// TwinCAT 3 PLC project CSVExample
// ProgramVersion: 3.1.0.8
// libraries:
//   Tc2_Math, * (Beckhoff Automation GmbH)
//   Tc2_Standard, * (Beckhoff Automation GmbH)
//   Tc2_System, * (Beckhoff Automation GmbH)
//   Tc2_Utilities, * (Beckhoff Automation GmbH)
//   Tc3_Module, * (Beckhoff Automation GmbH)
//   VisuDialogs, * (System)
//   Base Interfaces,newest,System
//   VisuSymbols,3.5.10.0,System
// project tree:
//   DUTs/ arr_rt.TcDUT (not stored), ENUM_BufferMgmt.TcDUT, ENUM_SeqSM.TcDUT, ST_CSV_Record.TcDUT (not stored)
//   DUTs/typ_FB_Debounce/ typFBDInOut.TcDUT (not stored), typFBDInput.TcDUT, typFBDOutput.TcDUT (not stored), typ_FBInt_Debounce.TcDUT
//   DUTs/typ_FB_DMX/ ENUM_IQ_OpMode.TcDUT (not stored), ENUM_I_ValRange.TcDUT (not stored), ENUM_I_Waveform.TcDUT, typDMXInOut.TcDUT (not stored), typDMXInput.TcDUT, typDMXOutput.TcDUT, typ_FBInt_DMX.TcDUT
//   / GlobalTextList.TcGTLO, PlcTask.TcTTO, Visualization Manager.TcVMO (not stored)
//   GVLs/ gc.TcGVL, gFB.TcGVL, GVL.TcGVL, g_ast.TcGVL
//   POUs/CSV read_write in binary mode/ P_BinaryModeRead.TcPOU, P_BinaryModeWrite.TcPOU (not stored)
//   POUs/CSV read_write in text mode/ P_TextModeRead.TcPOU (not stored), P_TextModeWrite.TcPOU (not stored)
//   POUs/ DMXTest.TcPOU, MAIN.TcPOU, P_ArgToConvExample.TcPOU, P_StringToConvExample.TcPOU
//   POUs/FunctionBlocks/ FB_DMX.TcPOU, FB_InputDebounce.TcPOU (not stored)
//   POUs/FunctionBlocks/HelperPRG/ InterfaceLink.TcPOU, IOParams.TcPOU
//   POUs/Functions/ f_to_Period.TcPOU, Map.TcPOU, MapClamp.TcPOU, SclByteDMX.TcPOU (not stored), SclBytePNP.TcPOU
//   VISUs/ Visualization.TcVIS
// real-time tasks:
//   TASK PlcTask: cycle T#10ms, priority 20, ADS port 350
// I/O:
//   DEVICE Device 1 (EtherCAT) (disabled), AmsNetId 192.168.1.208.2.1
//     Term 1 (EK1100) [EK1100 EtherCAT Coupler (2A E-Bus)]
//       Term 2 (EL6851) [EL6851 DMX Master]
//       Term 3 (EL1008) [EL1008 8Ch. Dig. Input 24V, 3ms]
//       Term 4 (EL1008) [EL1008 8Ch. Dig. Input 24V, 3ms]
//       Term 5 (EL1008) [EL1008 8Ch. Dig. Input 24V, 3ms]
//       Term 29 (EL1008) [EL1008 8Ch. Dig. Input 24V, 3ms]
//       Term 30 (EL1008) [EL1008 8Ch. Dig. Input 24V, 3ms]
//       Term 31 (EL1008) [EL1008 8Ch. Dig. Input 24V, 3ms]
//       Term 32 (EL1008) [EL1008 8Ch. Dig. Input 24V, 3ms]
//       Term 33 (EL1008) [EL1008 8Ch. Dig. Input 24V, 3ms]
//       Term 34 (EL1008) [EL1008 8Ch. Dig. Input 24V, 3ms]
//       Term 35 (EL1008) [EL1008 8Ch. Dig. Input 24V, 3ms]
//       Term 36 (EL1088) [EL1088 8Ch. Dig. Input 24V, 3ms, negative]
//       Term 37 (EL1088) [EL1088 8Ch. Dig. Input 24V, 3ms, negative]
//       Term 38 (EL1088) [EL1088 8Ch. Dig. Input 24V, 3ms, negative]
//       Term 39 (EL1088) [EL1088 8Ch. Dig. Input 24V, 3ms, negative]
//       Term 40 (EL1088) [EL1088 8Ch. Dig. Input 24V, 3ms, negative]
//       Term 41 (EL9410) [EL9410 E-Bus Power Supplier  (Diagnostics)]
//       Term 42 (EL1088) [EL1088 8Ch. Dig. Input 24V, 3ms, negative]
//       Term 43 (EL1088) [EL1088 8Ch. Dig. Input 24V, 3ms, negative]
//       Term 44 (EL1088) [EL1088 8Ch. Dig. Input 24V, 3ms, negative]
//       Term 45 (EL1088) [EL1088 8Ch. Dig. Input 24V, 3ms, negative]
//       Term 46 (EL1088) [EL1088 8Ch. Dig. Input 24V, 3ms, negative]
//       Term 47 (EL9011) [EL9011 End Terminal]
// variable links:
//   CSVExample/CSVExample Instance <-> Device 1 (EtherCAT)/Term 1 (EK1100)/Term 2 (EL6851)
//     PlcTask Outputs/g_ast.DMXHWOut[0] <-> DMX Channel 1-64/Channel 1
//     PlcTask Outputs/g_ast.DMXHWOut[100] <-> DMX Channel 65-128/Channel 101
//     PlcTask Outputs/g_ast.DMXHWOut[101] <-> DMX Channel 65-128/Channel 102
//     PlcTask Outputs/g_ast.DMXHWOut[102] <-> DMX Channel 65-128/Channel 103
//     PlcTask Outputs/g_ast.DMXHWOut[103] <-> DMX Channel 65-128/Channel 104
//     PlcTask Outputs/g_ast.DMXHWOut[104] <-> DMX Channel 65-128/Channel 105
//     PlcTask Outputs/g_ast.DMXHWOut[105] <-> DMX Channel 65-128/Channel 106
//     PlcTask Outputs/g_ast.DMXHWOut[106] <-> DMX Channel 65-128/Channel 107
//     PlcTask Outputs/g_ast.DMXHWOut[107] <-> DMX Channel 65-128/Channel 108
//     PlcTask Outputs/g_ast.DMXHWOut[108] <-> DMX Channel 65-128/Channel 109
//     PlcTask Outputs/g_ast.DMXHWOut[109] <-> DMX Channel 65-128/Channel 110
//     PlcTask Outputs/g_ast.DMXHWOut[10] <-> DMX Channel 1-64/Channel 11
//     PlcTask Outputs/g_ast.DMXHWOut[110] <-> DMX Channel 65-128/Channel 111
//     PlcTask Outputs/g_ast.DMXHWOut[111] <-> DMX Channel 65-128/Channel 112
//     PlcTask Outputs/g_ast.DMXHWOut[112] <-> DMX Channel 65-128/Channel 113
//     PlcTask Outputs/g_ast.DMXHWOut[113] <-> DMX Channel 65-128/Channel 114
//     PlcTask Outputs/g_ast.DMXHWOut[114] <-> DMX Channel 65-128/Channel 115
//     PlcTask Outputs/g_ast.DMXHWOut[115] <-> DMX Channel 65-128/Channel 116
//     PlcTask Outputs/g_ast.DMXHWOut[116] <-> DMX Channel 65-128/Channel 117
//     PlcTask Outputs/g_ast.DMXHWOut[117] <-> DMX Channel 65-128/Channel 118
//     PlcTask Outputs/g_ast.DMXHWOut[118] <-> DMX Channel 65-128/Channel 119
//     PlcTask Outputs/g_ast.DMXHWOut[119] <-> DMX Channel 65-128/Channel 120
//     PlcTask Outputs/g_ast.DMXHWOut[11] <-> DMX Channel 1-64/Channel 12
//     PlcTask Outputs/g_ast.DMXHWOut[120] <-> DMX Channel 65-128/Channel 121
//     PlcTask Outputs/g_ast.DMXHWOut[121] <-> DMX Channel 65-128/Channel 122
//     PlcTask Outputs/g_ast.DMXHWOut[122] <-> DMX Channel 65-128/Channel 123
//     PlcTask Outputs/g_ast.DMXHWOut[123] <-> DMX Channel 65-128/Channel 124
//     PlcTask Outputs/g_ast.DMXHWOut[124] <-> DMX Channel 65-128/Channel 125
//     PlcTask Outputs/g_ast.DMXHWOut[125] <-> DMX Channel 65-128/Channel 126
//     PlcTask Outputs/g_ast.DMXHWOut[126] <-> DMX Channel 65-128/Channel 127
//     PlcTask Outputs/g_ast.DMXHWOut[127] <-> DMX Channel 65-128/Channel 128
//     PlcTask Outputs/g_ast.DMXHWOut[128] <-> DMX Channel 129-192/Channel 129
//     PlcTask Outputs/g_ast.DMXHWOut[129] <-> DMX Channel 129-192/Channel 130
//     PlcTask Outputs/g_ast.DMXHWOut[12] <-> DMX Channel 1-64/Channel 13
//     PlcTask Outputs/g_ast.DMXHWOut[130] <-> DMX Channel 129-192/Channel 131
//     PlcTask Outputs/g_ast.DMXHWOut[131] <-> DMX Channel 129-192/Channel 132
//     PlcTask Outputs/g_ast.DMXHWOut[132] <-> DMX Channel 129-192/Channel 133
//     PlcTask Outputs/g_ast.DMXHWOut[133] <-> DMX Channel 129-192/Channel 134
//     PlcTask Outputs/g_ast.DMXHWOut[134] <-> DMX Channel 129-192/Channel 135
//     PlcTask Outputs/g_ast.DMXHWOut[135] <-> DMX Channel 129-192/Channel 136
//     PlcTask Outputs/g_ast.DMXHWOut[136] <-> DMX Channel 129-192/Channel 137
//     PlcTask Outputs/g_ast.DMXHWOut[137] <-> DMX Channel 129-192/Channel 138
//     PlcTask Outputs/g_ast.DMXHWOut[138] <-> DMX Channel 129-192/Channel 139
//     PlcTask Outputs/g_ast.DMXHWOut[139] <-> DMX Channel 129-192/Channel 140
//     PlcTask Outputs/g_ast.DMXHWOut[13] <-> DMX Channel 1-64/Channel 14
//     PlcTask Outputs/g_ast.DMXHWOut[140] <-> DMX Channel 129-192/Channel 141
//     PlcTask Outputs/g_ast.DMXHWOut[141] <-> DMX Channel 129-192/Channel 142
//     PlcTask Outputs/g_ast.DMXHWOut[142] <-> DMX Channel 129-192/Channel 143
//     PlcTask Outputs/g_ast.DMXHWOut[143] <-> DMX Channel 129-192/Channel 144
//     PlcTask Outputs/g_ast.DMXHWOut[144] <-> DMX Channel 129-192/Channel 145
//     PlcTask Outputs/g_ast.DMXHWOut[145] <-> DMX Channel 129-192/Channel 146
//     PlcTask Outputs/g_ast.DMXHWOut[146] <-> DMX Channel 129-192/Channel 147
//     PlcTask Outputs/g_ast.DMXHWOut[147] <-> DMX Channel 129-192/Channel 148
//     PlcTask Outputs/g_ast.DMXHWOut[148] <-> DMX Channel 129-192/Channel 149
//     PlcTask Outputs/g_ast.DMXHWOut[149] <-> DMX Channel 129-192/Channel 150
//     PlcTask Outputs/g_ast.DMXHWOut[14] <-> DMX Channel 1-64/Channel 15
//     PlcTask Outputs/g_ast.DMXHWOut[150] <-> DMX Channel 129-192/Channel 151
//     PlcTask Outputs/g_ast.DMXHWOut[151] <-> DMX Channel 129-192/Channel 152
//     PlcTask Outputs/g_ast.DMXHWOut[152] <-> DMX Channel 129-192/Channel 153
//     PlcTask Outputs/g_ast.DMXHWOut[153] <-> DMX Channel 129-192/Channel 154
//     PlcTask Outputs/g_ast.DMXHWOut[154] <-> DMX Channel 129-192/Channel 155
//     PlcTask Outputs/g_ast.DMXHWOut[155] <-> DMX Channel 129-192/Channel 156
//     PlcTask Outputs/g_ast.DMXHWOut[156] <-> DMX Channel 129-192/Channel 157
//     PlcTask Outputs/g_ast.DMXHWOut[157] <-> DMX Channel 129-192/Channel 158
//     PlcTask Outputs/g_ast.DMXHWOut[158] <-> DMX Channel 129-192/Channel 159
//     PlcTask Outputs/g_ast.DMXHWOut[159] <-> DMX Channel 129-192/Channel 160
//     PlcTask Outputs/g_ast.DMXHWOut[15] <-> DMX Channel 1-64/Channel 16
//     PlcTask Outputs/g_ast.DMXHWOut[160] <-> DMX Channel 129-192/Channel 161
//     PlcTask Outputs/g_ast.DMXHWOut[161] <-> DMX Channel 129-192/Channel 162
//     PlcTask Outputs/g_ast.DMXHWOut[162] <-> DMX Channel 129-192/Channel 163
//     PlcTask Outputs/g_ast.DMXHWOut[163] <-> DMX Channel 129-192/Channel 164
//     PlcTask Outputs/g_ast.DMXHWOut[164] <-> DMX Channel 129-192/Channel 165
//     PlcTask Outputs/g_ast.DMXHWOut[165] <-> DMX Channel 129-192/Channel 166
//     PlcTask Outputs/g_ast.DMXHWOut[166] <-> DMX Channel 129-192/Channel 167
//     PlcTask Outputs/g_ast.DMXHWOut[167] <-> DMX Channel 129-192/Channel 168
//     PlcTask Outputs/g_ast.DMXHWOut[168] <-> DMX Channel 129-192/Channel 169
//     PlcTask Outputs/g_ast.DMXHWOut[169] <-> DMX Channel 129-192/Channel 170
//     PlcTask Outputs/g_ast.DMXHWOut[16] <-> DMX Channel 1-64/Channel 17
//     PlcTask Outputs/g_ast.DMXHWOut[170] <-> DMX Channel 129-192/Channel 171
//     PlcTask Outputs/g_ast.DMXHWOut[171] <-> DMX Channel 129-192/Channel 172
//     PlcTask Outputs/g_ast.DMXHWOut[172] <-> DMX Channel 129-192/Channel 173
//     PlcTask Outputs/g_ast.DMXHWOut[173] <-> DMX Channel 129-192/Channel 174
//     PlcTask Outputs/g_ast.DMXHWOut[174] <-> DMX Channel 129-192/Channel 175
//     PlcTask Outputs/g_ast.DMXHWOut[175] <-> DMX Channel 129-192/Channel 176
//     PlcTask Outputs/g_ast.DMXHWOut[176] <-> DMX Channel 129-192/Channel 177
//     PlcTask Outputs/g_ast.DMXHWOut[177] <-> DMX Channel 129-192/Channel 178
//     PlcTask Outputs/g_ast.DMXHWOut[178] <-> DMX Channel 129-192/Channel 179
//     PlcTask Outputs/g_ast.DMXHWOut[179] <-> DMX Channel 129-192/Channel 180
//     PlcTask Outputs/g_ast.DMXHWOut[17] <-> DMX Channel 1-64/Channel 18
//     PlcTask Outputs/g_ast.DMXHWOut[180] <-> DMX Channel 129-192/Channel 181
//     PlcTask Outputs/g_ast.DMXHWOut[181] <-> DMX Channel 129-192/Channel 182
//     PlcTask Outputs/g_ast.DMXHWOut[182] <-> DMX Channel 129-192/Channel 183
//     PlcTask Outputs/g_ast.DMXHWOut[183] <-> DMX Channel 129-192/Channel 184
//     PlcTask Outputs/g_ast.DMXHWOut[184] <-> DMX Channel 129-192/Channel 185
//     PlcTask Outputs/g_ast.DMXHWOut[185] <-> DMX Channel 129-192/Channel 186
//     PlcTask Outputs/g_ast.DMXHWOut[186] <-> DMX Channel 129-192/Channel 187
//     PlcTask Outputs/g_ast.DMXHWOut[187] <-> DMX Channel 129-192/Channel 188
//     PlcTask Outputs/g_ast.DMXHWOut[188] <-> DMX Channel 129-192/Channel 189
//     PlcTask Outputs/g_ast.DMXHWOut[189] <-> DMX Channel 129-192/Channel 190
//     PlcTask Outputs/g_ast.DMXHWOut[18] <-> DMX Channel 1-64/Channel 19
//     PlcTask Outputs/g_ast.DMXHWOut[190] <-> DMX Channel 129-192/Channel 191
//     PlcTask Outputs/g_ast.DMXHWOut[191] <-> DMX Channel 129-192/Channel 192
//     PlcTask Outputs/g_ast.DMXHWOut[192] <-> DMX Channel 193-256/Channel 193
//     PlcTask Outputs/g_ast.DMXHWOut[193] <-> DMX Channel 193-256/Channel 194
//     PlcTask Outputs/g_ast.DMXHWOut[194] <-> DMX Channel 193-256/Channel 195
//     PlcTask Outputs/g_ast.DMXHWOut[195] <-> DMX Channel 193-256/Channel 196
//     PlcTask Outputs/g_ast.DMXHWOut[196] <-> DMX Channel 193-256/Channel 197
//     PlcTask Outputs/g_ast.DMXHWOut[197] <-> DMX Channel 193-256/Channel 198
//     PlcTask Outputs/g_ast.DMXHWOut[198] <-> DMX Channel 193-256/Channel 199
//     PlcTask Outputs/g_ast.DMXHWOut[199] <-> DMX Channel 193-256/Channel 200
//     PlcTask Outputs/g_ast.DMXHWOut[19] <-> DMX Channel 1-64/Channel 20
//     PlcTask Outputs/g_ast.DMXHWOut[1] <-> DMX Channel 1-64/Channel 2
//     PlcTask Outputs/g_ast.DMXHWOut[200] <-> DMX Channel 193-256/Channel 201
//     PlcTask Outputs/g_ast.DMXHWOut[201] <-> DMX Channel 193-256/Channel 202
//     PlcTask Outputs/g_ast.DMXHWOut[202] <-> DMX Channel 193-256/Channel 203
//     PlcTask Outputs/g_ast.DMXHWOut[203] <-> DMX Channel 193-256/Channel 204
//     PlcTask Outputs/g_ast.DMXHWOut[204] <-> DMX Channel 193-256/Channel 205
//     PlcTask Outputs/g_ast.DMXHWOut[205] <-> DMX Channel 193-256/Channel 206
//     PlcTask Outputs/g_ast.DMXHWOut[206] <-> DMX Channel 193-256/Channel 207
//     PlcTask Outputs/g_ast.DMXHWOut[207] <-> DMX Channel 193-256/Channel 208
//     PlcTask Outputs/g_ast.DMXHWOut[208] <-> DMX Channel 193-256/Channel 209
//     PlcTask Outputs/g_ast.DMXHWOut[209] <-> DMX Channel 193-256/Channel 210
//     PlcTask Outputs/g_ast.DMXHWOut[20] <-> DMX Channel 1-64/Channel 21
//     PlcTask Outputs/g_ast.DMXHWOut[210] <-> DMX Channel 193-256/Channel 211
//     PlcTask Outputs/g_ast.DMXHWOut[211] <-> DMX Channel 193-256/Channel 212
//     PlcTask Outputs/g_ast.DMXHWOut[212] <-> DMX Channel 193-256/Channel 213
//     PlcTask Outputs/g_ast.DMXHWOut[213] <-> DMX Channel 193-256/Channel 214
//     PlcTask Outputs/g_ast.DMXHWOut[214] <-> DMX Channel 193-256/Channel 215
//     PlcTask Outputs/g_ast.DMXHWOut[215] <-> DMX Channel 193-256/Channel 216
//     PlcTask Outputs/g_ast.DMXHWOut[216] <-> DMX Channel 193-256/Channel 217
//     PlcTask Outputs/g_ast.DMXHWOut[217] <-> DMX Channel 193-256/Channel 218
//     PlcTask Outputs/g_ast.DMXHWOut[218] <-> DMX Channel 193-256/Channel 219
//     PlcTask Outputs/g_ast.DMXHWOut[219] <-> DMX Channel 193-256/Channel 220
//     PlcTask Outputs/g_ast.DMXHWOut[21] <-> DMX Channel 1-64/Channel 22
//     PlcTask Outputs/g_ast.DMXHWOut[220] <-> DMX Channel 193-256/Channel 221
//     PlcTask Outputs/g_ast.DMXHWOut[221] <-> DMX Channel 193-256/Channel 222
//     PlcTask Outputs/g_ast.DMXHWOut[222] <-> DMX Channel 193-256/Channel 223
//     PlcTask Outputs/g_ast.DMXHWOut[223] <-> DMX Channel 193-256/Channel 224
//     PlcTask Outputs/g_ast.DMXHWOut[224] <-> DMX Channel 193-256/Channel 225
//     PlcTask Outputs/g_ast.DMXHWOut[225] <-> DMX Channel 193-256/Channel 226
//     PlcTask Outputs/g_ast.DMXHWOut[226] <-> DMX Channel 193-256/Channel 227
//     PlcTask Outputs/g_ast.DMXHWOut[227] <-> DMX Channel 193-256/Channel 228
//     PlcTask Outputs/g_ast.DMXHWOut[228] <-> DMX Channel 193-256/Channel 229
//     PlcTask Outputs/g_ast.DMXHWOut[229] <-> DMX Channel 193-256/Channel 230
//     PlcTask Outputs/g_ast.DMXHWOut[22] <-> DMX Channel 1-64/Channel 23
//     PlcTask Outputs/g_ast.DMXHWOut[230] <-> DMX Channel 193-256/Channel 231
//     PlcTask Outputs/g_ast.DMXHWOut[231] <-> DMX Channel 193-256/Channel 232
//     PlcTask Outputs/g_ast.DMXHWOut[232] <-> DMX Channel 193-256/Channel 233
//     PlcTask Outputs/g_ast.DMXHWOut[233] <-> DMX Channel 193-256/Channel 234
//     PlcTask Outputs/g_ast.DMXHWOut[234] <-> DMX Channel 193-256/Channel 235
//     PlcTask Outputs/g_ast.DMXHWOut[235] <-> DMX Channel 193-256/Channel 236
//     PlcTask Outputs/g_ast.DMXHWOut[236] <-> DMX Channel 193-256/Channel 237
//     PlcTask Outputs/g_ast.DMXHWOut[237] <-> DMX Channel 193-256/Channel 238
//     PlcTask Outputs/g_ast.DMXHWOut[238] <-> DMX Channel 193-256/Channel 239
//     PlcTask Outputs/g_ast.DMXHWOut[239] <-> DMX Channel 193-256/Channel 240
//     PlcTask Outputs/g_ast.DMXHWOut[23] <-> DMX Channel 1-64/Channel 24
//     PlcTask Outputs/g_ast.DMXHWOut[240] <-> DMX Channel 193-256/Channel 241
//     PlcTask Outputs/g_ast.DMXHWOut[241] <-> DMX Channel 193-256/Channel 242
//     PlcTask Outputs/g_ast.DMXHWOut[242] <-> DMX Channel 193-256/Channel 243
//     PlcTask Outputs/g_ast.DMXHWOut[243] <-> DMX Channel 193-256/Channel 244
//     PlcTask Outputs/g_ast.DMXHWOut[244] <-> DMX Channel 193-256/Channel 245
//     PlcTask Outputs/g_ast.DMXHWOut[245] <-> DMX Channel 193-256/Channel 246
//     PlcTask Outputs/g_ast.DMXHWOut[246] <-> DMX Channel 193-256/Channel 247
//     PlcTask Outputs/g_ast.DMXHWOut[247] <-> DMX Channel 193-256/Channel 248
//     PlcTask Outputs/g_ast.DMXHWOut[248] <-> DMX Channel 193-256/Channel 249
//     PlcTask Outputs/g_ast.DMXHWOut[249] <-> DMX Channel 193-256/Channel 250
//     PlcTask Outputs/g_ast.DMXHWOut[24] <-> DMX Channel 1-64/Channel 25
//     PlcTask Outputs/g_ast.DMXHWOut[250] <-> DMX Channel 193-256/Channel 251
//     PlcTask Outputs/g_ast.DMXHWOut[251] <-> DMX Channel 193-256/Channel 252
//     PlcTask Outputs/g_ast.DMXHWOut[252] <-> DMX Channel 193-256/Channel 253
//     PlcTask Outputs/g_ast.DMXHWOut[253] <-> DMX Channel 193-256/Channel 254
//     PlcTask Outputs/g_ast.DMXHWOut[254] <-> DMX Channel 193-256/Channel 255
//     PlcTask Outputs/g_ast.DMXHWOut[255] <-> DMX Channel 193-256/Channel 256
//     PlcTask Outputs/g_ast.DMXHWOut[256] <-> DMX Channel 257-320/Channel 257
//     PlcTask Outputs/g_ast.DMXHWOut[257] <-> DMX Channel 257-320/Channel 258
//     PlcTask Outputs/g_ast.DMXHWOut[258] <-> DMX Channel 257-320/Channel 259
//     PlcTask Outputs/g_ast.DMXHWOut[259] <-> DMX Channel 257-320/Channel 260
//     PlcTask Outputs/g_ast.DMXHWOut[25] <-> DMX Channel 1-64/Channel 26
//     PlcTask Outputs/g_ast.DMXHWOut[260] <-> DMX Channel 257-320/Channel 261
//     PlcTask Outputs/g_ast.DMXHWOut[261] <-> DMX Channel 257-320/Channel 262
//     PlcTask Outputs/g_ast.DMXHWOut[262] <-> DMX Channel 257-320/Channel 263
//     PlcTask Outputs/g_ast.DMXHWOut[263] <-> DMX Channel 257-320/Channel 264
//     PlcTask Outputs/g_ast.DMXHWOut[264] <-> DMX Channel 257-320/Channel 265
//     PlcTask Outputs/g_ast.DMXHWOut[265] <-> DMX Channel 257-320/Channel 266
//     PlcTask Outputs/g_ast.DMXHWOut[266] <-> DMX Channel 257-320/Channel 267
//     PlcTask Outputs/g_ast.DMXHWOut[267] <-> DMX Channel 257-320/Channel 268
//     PlcTask Outputs/g_ast.DMXHWOut[268] <-> DMX Channel 257-320/Channel 269
//     PlcTask Outputs/g_ast.DMXHWOut[269] <-> DMX Channel 257-320/Channel 270
//     PlcTask Outputs/g_ast.DMXHWOut[26] <-> DMX Channel 1-64/Channel 27
//     PlcTask Outputs/g_ast.DMXHWOut[270] <-> DMX Channel 257-320/Channel 271
//     PlcTask Outputs/g_ast.DMXHWOut[271] <-> DMX Channel 257-320/Channel 272
//     PlcTask Outputs/g_ast.DMXHWOut[272] <-> DMX Channel 257-320/Channel 273
//     PlcTask Outputs/g_ast.DMXHWOut[273] <-> DMX Channel 257-320/Channel 274
//     PlcTask Outputs/g_ast.DMXHWOut[274] <-> DMX Channel 257-320/Channel 275
//     PlcTask Outputs/g_ast.DMXHWOut[275] <-> DMX Channel 257-320/Channel 276
//     PlcTask Outputs/g_ast.DMXHWOut[276] <-> DMX Channel 257-320/Channel 277
//     PlcTask Outputs/g_ast.DMXHWOut[277] <-> DMX Channel 257-320/Channel 278
//     PlcTask Outputs/g_ast.DMXHWOut[278] <-> DMX Channel 257-320/Channel 279
//     PlcTask Outputs/g_ast.DMXHWOut[279] <-> DMX Channel 257-320/Channel 280
//     PlcTask Outputs/g_ast.DMXHWOut[27] <-> DMX Channel 1-64/Channel 28
//     PlcTask Outputs/g_ast.DMXHWOut[280] <-> DMX Channel 257-320/Channel 281
//     PlcTask Outputs/g_ast.DMXHWOut[281] <-> DMX Channel 257-320/Channel 282
//     PlcTask Outputs/g_ast.DMXHWOut[282] <-> DMX Channel 257-320/Channel 283
//     PlcTask Outputs/g_ast.DMXHWOut[283] <-> DMX Channel 257-320/Channel 284
//     PlcTask Outputs/g_ast.DMXHWOut[284] <-> DMX Channel 257-320/Channel 285
//     PlcTask Outputs/g_ast.DMXHWOut[285] <-> DMX Channel 257-320/Channel 286
//     PlcTask Outputs/g_ast.DMXHWOut[286] <-> DMX Channel 257-320/Channel 287
//     PlcTask Outputs/g_ast.DMXHWOut[287] <-> DMX Channel 257-320/Channel 288
//     PlcTask Outputs/g_ast.DMXHWOut[288] <-> DMX Channel 257-320/Channel 289
//     PlcTask Outputs/g_ast.DMXHWOut[289] <-> DMX Channel 257-320/Channel 290
//     PlcTask Outputs/g_ast.DMXHWOut[28] <-> DMX Channel 1-64/Channel 29
//     PlcTask Outputs/g_ast.DMXHWOut[290] <-> DMX Channel 257-320/Channel 291
//     PlcTask Outputs/g_ast.DMXHWOut[291] <-> DMX Channel 257-320/Channel 292
//     PlcTask Outputs/g_ast.DMXHWOut[292] <-> DMX Channel 257-320/Channel 293
//     PlcTask Outputs/g_ast.DMXHWOut[293] <-> DMX Channel 257-320/Channel 294
//     PlcTask Outputs/g_ast.DMXHWOut[294] <-> DMX Channel 257-320/Channel 295
//     PlcTask Outputs/g_ast.DMXHWOut[295] <-> DMX Channel 257-320/Channel 296
//     PlcTask Outputs/g_ast.DMXHWOut[296] <-> DMX Channel 257-320/Channel 297
//     PlcTask Outputs/g_ast.DMXHWOut[297] <-> DMX Channel 257-320/Channel 298
//     PlcTask Outputs/g_ast.DMXHWOut[298] <-> DMX Channel 257-320/Channel 299
//     PlcTask Outputs/g_ast.DMXHWOut[299] <-> DMX Channel 257-320/Channel 300
//     PlcTask Outputs/g_ast.DMXHWOut[29] <-> DMX Channel 1-64/Channel 30
//     PlcTask Outputs/g_ast.DMXHWOut[2] <-> DMX Channel 1-64/Channel 3
//     PlcTask Outputs/g_ast.DMXHWOut[300] <-> DMX Channel 257-320/Channel 301
//     PlcTask Outputs/g_ast.DMXHWOut[301] <-> DMX Channel 257-320/Channel 302
//     PlcTask Outputs/g_ast.DMXHWOut[302] <-> DMX Channel 257-320/Channel 303
//     PlcTask Outputs/g_ast.DMXHWOut[303] <-> DMX Channel 257-320/Channel 304
//     PlcTask Outputs/g_ast.DMXHWOut[304] <-> DMX Channel 257-320/Channel 305
//     PlcTask Outputs/g_ast.DMXHWOut[305] <-> DMX Channel 257-320/Channel 306
//     PlcTask Outputs/g_ast.DMXHWOut[306] <-> DMX Channel 257-320/Channel 307
//     PlcTask Outputs/g_ast.DMXHWOut[307] <-> DMX Channel 257-320/Channel 308
//     PlcTask Outputs/g_ast.DMXHWOut[308] <-> DMX Channel 257-320/Channel 309
//     PlcTask Outputs/g_ast.DMXHWOut[309] <-> DMX Channel 257-320/Channel 310
//     PlcTask Outputs/g_ast.DMXHWOut[30] <-> DMX Channel 1-64/Channel 31
//     PlcTask Outputs/g_ast.DMXHWOut[310] <-> DMX Channel 257-320/Channel 311
//     PlcTask Outputs/g_ast.DMXHWOut[311] <-> DMX Channel 257-320/Channel 312
//     PlcTask Outputs/g_ast.DMXHWOut[312] <-> DMX Channel 257-320/Channel 313
//     PlcTask Outputs/g_ast.DMXHWOut[313] <-> DMX Channel 257-320/Channel 314
//     PlcTask Outputs/g_ast.DMXHWOut[314] <-> DMX Channel 257-320/Channel 315
//     PlcTask Outputs/g_ast.DMXHWOut[315] <-> DMX Channel 257-320/Channel 316
//     PlcTask Outputs/g_ast.DMXHWOut[316] <-> DMX Channel 257-320/Channel 317
//     PlcTask Outputs/g_ast.DMXHWOut[317] <-> DMX Channel 257-320/Channel 318
//     PlcTask Outputs/g_ast.DMXHWOut[318] <-> DMX Channel 257-320/Channel 319
//     PlcTask Outputs/g_ast.DMXHWOut[319] <-> DMX Channel 257-320/Channel 320
//     PlcTask Outputs/g_ast.DMXHWOut[31] <-> DMX Channel 1-64/Channel 32
//     PlcTask Outputs/g_ast.DMXHWOut[320] <-> DMX Channel 321-384/Channel 321
//     PlcTask Outputs/g_ast.DMXHWOut[321] <-> DMX Channel 321-384/Channel 322
//     PlcTask Outputs/g_ast.DMXHWOut[322] <-> DMX Channel 321-384/Channel 323
//     PlcTask Outputs/g_ast.DMXHWOut[323] <-> DMX Channel 321-384/Channel 324
//     PlcTask Outputs/g_ast.DMXHWOut[324] <-> DMX Channel 321-384/Channel 325
//     PlcTask Outputs/g_ast.DMXHWOut[325] <-> DMX Channel 321-384/Channel 326
//     PlcTask Outputs/g_ast.DMXHWOut[326] <-> DMX Channel 321-384/Channel 327
//     PlcTask Outputs/g_ast.DMXHWOut[327] <-> DMX Channel 321-384/Channel 328
//     PlcTask Outputs/g_ast.DMXHWOut[328] <-> DMX Channel 321-384/Channel 329
//     PlcTask Outputs/g_ast.DMXHWOut[329] <-> DMX Channel 321-384/Channel 330
//     PlcTask Outputs/g_ast.DMXHWOut[32] <-> DMX Channel 1-64/Channel 33
//     PlcTask Outputs/g_ast.DMXHWOut[330] <-> DMX Channel 321-384/Channel 331
//     PlcTask Outputs/g_ast.DMXHWOut[331] <-> DMX Channel 321-384/Channel 332
//     PlcTask Outputs/g_ast.DMXHWOut[332] <-> DMX Channel 321-384/Channel 333
//     PlcTask Outputs/g_ast.DMXHWOut[333] <-> DMX Channel 321-384/Channel 334
//     PlcTask Outputs/g_ast.DMXHWOut[334] <-> DMX Channel 321-384/Channel 335
//     PlcTask Outputs/g_ast.DMXHWOut[335] <-> DMX Channel 321-384/Channel 336
//     PlcTask Outputs/g_ast.DMXHWOut[336] <-> DMX Channel 321-384/Channel 337
//     PlcTask Outputs/g_ast.DMXHWOut[337] <-> DMX Channel 321-384/Channel 338
//     PlcTask Outputs/g_ast.DMXHWOut[338] <-> DMX Channel 321-384/Channel 339
//     PlcTask Outputs/g_ast.DMXHWOut[339] <-> DMX Channel 321-384/Channel 340
//     PlcTask Outputs/g_ast.DMXHWOut[33] <-> DMX Channel 1-64/Channel 34
//     PlcTask Outputs/g_ast.DMXHWOut[340] <-> DMX Channel 321-384/Channel 341
//     PlcTask Outputs/g_ast.DMXHWOut[341] <-> DMX Channel 321-384/Channel 342
//     PlcTask Outputs/g_ast.DMXHWOut[342] <-> DMX Channel 321-384/Channel 343
//     PlcTask Outputs/g_ast.DMXHWOut[343] <-> DMX Channel 321-384/Channel 344
//     PlcTask Outputs/g_ast.DMXHWOut[344] <-> DMX Channel 321-384/Channel 345
//     PlcTask Outputs/g_ast.DMXHWOut[345] <-> DMX Channel 321-384/Channel 346
//     PlcTask Outputs/g_ast.DMXHWOut[346] <-> DMX Channel 321-384/Channel 347
//     PlcTask Outputs/g_ast.DMXHWOut[347] <-> DMX Channel 321-384/Channel 348
//     PlcTask Outputs/g_ast.DMXHWOut[348] <-> DMX Channel 321-384/Channel 349
//     PlcTask Outputs/g_ast.DMXHWOut[349] <-> DMX Channel 321-384/Channel 350
//     PlcTask Outputs/g_ast.DMXHWOut[34] <-> DMX Channel 1-64/Channel 35
//     PlcTask Outputs/g_ast.DMXHWOut[350] <-> DMX Channel 321-384/Channel 351
//     PlcTask Outputs/g_ast.DMXHWOut[351] <-> DMX Channel 321-384/Channel 352
//     PlcTask Outputs/g_ast.DMXHWOut[352] <-> DMX Channel 321-384/Channel 353
//     PlcTask Outputs/g_ast.DMXHWOut[353] <-> DMX Channel 321-384/Channel 354
//     PlcTask Outputs/g_ast.DMXHWOut[354] <-> DMX Channel 321-384/Channel 355
//     PlcTask Outputs/g_ast.DMXHWOut[355] <-> DMX Channel 321-384/Channel 356
//     PlcTask Outputs/g_ast.DMXHWOut[356] <-> DMX Channel 321-384/Channel 357
//     PlcTask Outputs/g_ast.DMXHWOut[357] <-> DMX Channel 321-384/Channel 358
//     PlcTask Outputs/g_ast.DMXHWOut[358] <-> DMX Channel 321-384/Channel 359
//     PlcTask Outputs/g_ast.DMXHWOut[359] <-> DMX Channel 321-384/Channel 360
//     PlcTask Outputs/g_ast.DMXHWOut[35] <-> DMX Channel 1-64/Channel 36
//     PlcTask Outputs/g_ast.DMXHWOut[360] <-> DMX Channel 321-384/Channel 361
//     PlcTask Outputs/g_ast.DMXHWOut[361] <-> DMX Channel 321-384/Channel 362
//     PlcTask Outputs/g_ast.DMXHWOut[362] <-> DMX Channel 321-384/Channel 363
//     PlcTask Outputs/g_ast.DMXHWOut[363] <-> DMX Channel 321-384/Channel 364
//     PlcTask Outputs/g_ast.DMXHWOut[364] <-> DMX Channel 321-384/Channel 365
//     PlcTask Outputs/g_ast.DMXHWOut[365] <-> DMX Channel 321-384/Channel 366
//     PlcTask Outputs/g_ast.DMXHWOut[366] <-> DMX Channel 321-384/Channel 367
//     PlcTask Outputs/g_ast.DMXHWOut[367] <-> DMX Channel 321-384/Channel 368
//     PlcTask Outputs/g_ast.DMXHWOut[368] <-> DMX Channel 321-384/Channel 369
//     PlcTask Outputs/g_ast.DMXHWOut[369] <-> DMX Channel 321-384/Channel 370
//     PlcTask Outputs/g_ast.DMXHWOut[36] <-> DMX Channel 1-64/Channel 37
//     PlcTask Outputs/g_ast.DMXHWOut[370] <-> DMX Channel 321-384/Channel 371
//     PlcTask Outputs/g_ast.DMXHWOut[371] <-> DMX Channel 321-384/Channel 372
//     PlcTask Outputs/g_ast.DMXHWOut[372] <-> DMX Channel 321-384/Channel 373
//     PlcTask Outputs/g_ast.DMXHWOut[373] <-> DMX Channel 321-384/Channel 374
//     PlcTask Outputs/g_ast.DMXHWOut[374] <-> DMX Channel 321-384/Channel 375
//     PlcTask Outputs/g_ast.DMXHWOut[375] <-> DMX Channel 321-384/Channel 376
//     PlcTask Outputs/g_ast.DMXHWOut[376] <-> DMX Channel 321-384/Channel 377
//     PlcTask Outputs/g_ast.DMXHWOut[377] <-> DMX Channel 321-384/Channel 378
//     PlcTask Outputs/g_ast.DMXHWOut[378] <-> DMX Channel 321-384/Channel 379
//     PlcTask Outputs/g_ast.DMXHWOut[379] <-> DMX Channel 321-384/Channel 380
//     PlcTask Outputs/g_ast.DMXHWOut[37] <-> DMX Channel 1-64/Channel 38
//     PlcTask Outputs/g_ast.DMXHWOut[380] <-> DMX Channel 321-384/Channel 381
//     PlcTask Outputs/g_ast.DMXHWOut[381] <-> DMX Channel 321-384/Channel 382
//     PlcTask Outputs/g_ast.DMXHWOut[382] <-> DMX Channel 321-384/Channel 383
//     PlcTask Outputs/g_ast.DMXHWOut[383] <-> DMX Channel 321-384/Channel 384
//     PlcTask Outputs/g_ast.DMXHWOut[384] <-> DMX Channel 385-448/Channel 385
//     PlcTask Outputs/g_ast.DMXHWOut[385] <-> DMX Channel 385-448/Channel 386
//     PlcTask Outputs/g_ast.DMXHWOut[386] <-> DMX Channel 385-448/Channel 387
//     PlcTask Outputs/g_ast.DMXHWOut[387] <-> DMX Channel 385-448/Channel 388
//     PlcTask Outputs/g_ast.DMXHWOut[388] <-> DMX Channel 385-448/Channel 389
//     PlcTask Outputs/g_ast.DMXHWOut[389] <-> DMX Channel 385-448/Channel 390
//     PlcTask Outputs/g_ast.DMXHWOut[38] <-> DMX Channel 1-64/Channel 39
//     PlcTask Outputs/g_ast.DMXHWOut[390] <-> DMX Channel 385-448/Channel 391
//     PlcTask Outputs/g_ast.DMXHWOut[391] <-> DMX Channel 385-448/Channel 392
//     PlcTask Outputs/g_ast.DMXHWOut[392] <-> DMX Channel 385-448/Channel 393
//     PlcTask Outputs/g_ast.DMXHWOut[393] <-> DMX Channel 385-448/Channel 394
//     PlcTask Outputs/g_ast.DMXHWOut[394] <-> DMX Channel 385-448/Channel 395
//     PlcTask Outputs/g_ast.DMXHWOut[395] <-> DMX Channel 385-448/Channel 396
//     PlcTask Outputs/g_ast.DMXHWOut[396] <-> DMX Channel 385-448/Channel 397
//     PlcTask Outputs/g_ast.DMXHWOut[397] <-> DMX Channel 385-448/Channel 398
//     PlcTask Outputs/g_ast.DMXHWOut[398] <-> DMX Channel 385-448/Channel 399
//     PlcTask Outputs/g_ast.DMXHWOut[399] <-> DMX Channel 385-448/Channel 400
//     PlcTask Outputs/g_ast.DMXHWOut[39] <-> DMX Channel 1-64/Channel 40
//     PlcTask Outputs/g_ast.DMXHWOut[3] <-> DMX Channel 1-64/Channel 4
//     PlcTask Outputs/g_ast.DMXHWOut[400] <-> DMX Channel 385-448/Channel 401
//     PlcTask Outputs/g_ast.DMXHWOut[401] <-> DMX Channel 385-448/Channel 402
//     PlcTask Outputs/g_ast.DMXHWOut[402] <-> DMX Channel 385-448/Channel 403
//     PlcTask Outputs/g_ast.DMXHWOut[403] <-> DMX Channel 385-448/Channel 404
//     PlcTask Outputs/g_ast.DMXHWOut[404] <-> DMX Channel 385-448/Channel 405
//     PlcTask Outputs/g_ast.DMXHWOut[405] <-> DMX Channel 385-448/Channel 406
//     PlcTask Outputs/g_ast.DMXHWOut[406] <-> DMX Channel 385-448/Channel 407
//     PlcTask Outputs/g_ast.DMXHWOut[407] <-> DMX Channel 385-448/Channel 408
//     PlcTask Outputs/g_ast.DMXHWOut[408] <-> DMX Channel 385-448/Channel 409
//     PlcTask Outputs/g_ast.DMXHWOut[409] <-> DMX Channel 385-448/Channel 410
//     PlcTask Outputs/g_ast.DMXHWOut[40] <-> DMX Channel 1-64/Channel 41
//     PlcTask Outputs/g_ast.DMXHWOut[410] <-> DMX Channel 385-448/Channel 411
//     PlcTask Outputs/g_ast.DMXHWOut[411] <-> DMX Channel 385-448/Channel 412
//     PlcTask Outputs/g_ast.DMXHWOut[412] <-> DMX Channel 385-448/Channel 413
//     PlcTask Outputs/g_ast.DMXHWOut[413] <-> DMX Channel 385-448/Channel 414
//     PlcTask Outputs/g_ast.DMXHWOut[414] <-> DMX Channel 385-448/Channel 415
//     PlcTask Outputs/g_ast.DMXHWOut[415] <-> DMX Channel 385-448/Channel 416
//     PlcTask Outputs/g_ast.DMXHWOut[416] <-> DMX Channel 385-448/Channel 417
//     PlcTask Outputs/g_ast.DMXHWOut[417] <-> DMX Channel 385-448/Channel 418
//     PlcTask Outputs/g_ast.DMXHWOut[418] <-> DMX Channel 385-448/Channel 419
//     PlcTask Outputs/g_ast.DMXHWOut[419] <-> DMX Channel 385-448/Channel 420
//     PlcTask Outputs/g_ast.DMXHWOut[41] <-> DMX Channel 1-64/Channel 42
//     PlcTask Outputs/g_ast.DMXHWOut[420] <-> DMX Channel 385-448/Channel 421
//     PlcTask Outputs/g_ast.DMXHWOut[421] <-> DMX Channel 385-448/Channel 422
//     PlcTask Outputs/g_ast.DMXHWOut[422] <-> DMX Channel 385-448/Channel 423
//     PlcTask Outputs/g_ast.DMXHWOut[423] <-> DMX Channel 385-448/Channel 424
//     PlcTask Outputs/g_ast.DMXHWOut[424] <-> DMX Channel 385-448/Channel 425
//     PlcTask Outputs/g_ast.DMXHWOut[425] <-> DMX Channel 385-448/Channel 426
//     PlcTask Outputs/g_ast.DMXHWOut[426] <-> DMX Channel 385-448/Channel 427
//     PlcTask Outputs/g_ast.DMXHWOut[427] <-> DMX Channel 385-448/Channel 428
//     PlcTask Outputs/g_ast.DMXHWOut[428] <-> DMX Channel 385-448/Channel 429
//     PlcTask Outputs/g_ast.DMXHWOut[429] <-> DMX Channel 385-448/Channel 430
//     PlcTask Outputs/g_ast.DMXHWOut[42] <-> DMX Channel 1-64/Channel 43
//     PlcTask Outputs/g_ast.DMXHWOut[430] <-> DMX Channel 385-448/Channel 431
//     PlcTask Outputs/g_ast.DMXHWOut[431] <-> DMX Channel 385-448/Channel 432
//     PlcTask Outputs/g_ast.DMXHWOut[432] <-> DMX Channel 385-448/Channel 433
//     PlcTask Outputs/g_ast.DMXHWOut[433] <-> DMX Channel 385-448/Channel 434
//     PlcTask Outputs/g_ast.DMXHWOut[434] <-> DMX Channel 385-448/Channel 435
//     PlcTask Outputs/g_ast.DMXHWOut[435] <-> DMX Channel 385-448/Channel 436
//     PlcTask Outputs/g_ast.DMXHWOut[436] <-> DMX Channel 385-448/Channel 437
//     PlcTask Outputs/g_ast.DMXHWOut[437] <-> DMX Channel 385-448/Channel 438
//     PlcTask Outputs/g_ast.DMXHWOut[438] <-> DMX Channel 385-448/Channel 439
//     PlcTask Outputs/g_ast.DMXHWOut[439] <-> DMX Channel 385-448/Channel 440
//     PlcTask Outputs/g_ast.DMXHWOut[43] <-> DMX Channel 1-64/Channel 44
//     PlcTask Outputs/g_ast.DMXHWOut[440] <-> DMX Channel 385-448/Channel 441
//     PlcTask Outputs/g_ast.DMXHWOut[441] <-> DMX Channel 385-448/Channel 442
//     PlcTask Outputs/g_ast.DMXHWOut[442] <-> DMX Channel 385-448/Channel 443
//     PlcTask Outputs/g_ast.DMXHWOut[443] <-> DMX Channel 385-448/Channel 444
//     PlcTask Outputs/g_ast.DMXHWOut[444] <-> DMX Channel 385-448/Channel 445
//     PlcTask Outputs/g_ast.DMXHWOut[445] <-> DMX Channel 385-448/Channel 446
//     PlcTask Outputs/g_ast.DMXHWOut[446] <-> DMX Channel 385-448/Channel 447
//     PlcTask Outputs/g_ast.DMXHWOut[447] <-> DMX Channel 385-448/Channel 448
//     PlcTask Outputs/g_ast.DMXHWOut[448] <-> DMX Channel 449-512/Channel 449
//     PlcTask Outputs/g_ast.DMXHWOut[449] <-> DMX Channel 449-512/Channel 450
//     PlcTask Outputs/g_ast.DMXHWOut[44] <-> DMX Channel 1-64/Channel 45
//     PlcTask Outputs/g_ast.DMXHWOut[450] <-> DMX Channel 449-512/Channel 451
//     PlcTask Outputs/g_ast.DMXHWOut[451] <-> DMX Channel 449-512/Channel 452
//     PlcTask Outputs/g_ast.DMXHWOut[452] <-> DMX Channel 449-512/Channel 453
//     PlcTask Outputs/g_ast.DMXHWOut[453] <-> DMX Channel 449-512/Channel 454
//     PlcTask Outputs/g_ast.DMXHWOut[454] <-> DMX Channel 449-512/Channel 455
//     PlcTask Outputs/g_ast.DMXHWOut[455] <-> DMX Channel 449-512/Channel 456
//     PlcTask Outputs/g_ast.DMXHWOut[456] <-> DMX Channel 449-512/Channel 457
//     PlcTask Outputs/g_ast.DMXHWOut[457] <-> DMX Channel 449-512/Channel 458
//     PlcTask Outputs/g_ast.DMXHWOut[458] <-> DMX Channel 449-512/Channel 459
//     PlcTask Outputs/g_ast.DMXHWOut[459] <-> DMX Channel 449-512/Channel 460
//     PlcTask Outputs/g_ast.DMXHWOut[45] <-> DMX Channel 1-64/Channel 46
//     PlcTask Outputs/g_ast.DMXHWOut[460] <-> DMX Channel 449-512/Channel 461
//     PlcTask Outputs/g_ast.DMXHWOut[461] <-> DMX Channel 449-512/Channel 462
//     PlcTask Outputs/g_ast.DMXHWOut[462] <-> DMX Channel 449-512/Channel 463
//     PlcTask Outputs/g_ast.DMXHWOut[463] <-> DMX Channel 449-512/Channel 464
//     PlcTask Outputs/g_ast.DMXHWOut[464] <-> DMX Channel 449-512/Channel 465
//     PlcTask Outputs/g_ast.DMXHWOut[465] <-> DMX Channel 449-512/Channel 466
//     PlcTask Outputs/g_ast.DMXHWOut[466] <-> DMX Channel 449-512/Channel 467
//     PlcTask Outputs/g_ast.DMXHWOut[467] <-> DMX Channel 449-512/Channel 468
//     PlcTask Outputs/g_ast.DMXHWOut[468] <-> DMX Channel 449-512/Channel 469
//     PlcTask Outputs/g_ast.DMXHWOut[469] <-> DMX Channel 449-512/Channel 470
//     PlcTask Outputs/g_ast.DMXHWOut[46] <-> DMX Channel 1-64/Channel 47
//     PlcTask Outputs/g_ast.DMXHWOut[470] <-> DMX Channel 449-512/Channel 471
//     PlcTask Outputs/g_ast.DMXHWOut[471] <-> DMX Channel 449-512/Channel 472
//     PlcTask Outputs/g_ast.DMXHWOut[472] <-> DMX Channel 449-512/Channel 473
//     PlcTask Outputs/g_ast.DMXHWOut[473] <-> DMX Channel 449-512/Channel 474
//     PlcTask Outputs/g_ast.DMXHWOut[474] <-> DMX Channel 449-512/Channel 475
//     PlcTask Outputs/g_ast.DMXHWOut[475] <-> DMX Channel 449-512/Channel 476
//     PlcTask Outputs/g_ast.DMXHWOut[476] <-> DMX Channel 449-512/Channel 477
//     PlcTask Outputs/g_ast.DMXHWOut[477] <-> DMX Channel 449-512/Channel 478
//     PlcTask Outputs/g_ast.DMXHWOut[478] <-> DMX Channel 449-512/Channel 479
//     PlcTask Outputs/g_ast.DMXHWOut[479] <-> DMX Channel 449-512/Channel 480
//     PlcTask Outputs/g_ast.DMXHWOut[47] <-> DMX Channel 1-64/Channel 48
//     PlcTask Outputs/g_ast.DMXHWOut[480] <-> DMX Channel 449-512/Channel 481
//     PlcTask Outputs/g_ast.DMXHWOut[481] <-> DMX Channel 449-512/Channel 482
//     PlcTask Outputs/g_ast.DMXHWOut[482] <-> DMX Channel 449-512/Channel 483
//     PlcTask Outputs/g_ast.DMXHWOut[483] <-> DMX Channel 449-512/Channel 484
//     PlcTask Outputs/g_ast.DMXHWOut[484] <-> DMX Channel 449-512/Channel 485
//     PlcTask Outputs/g_ast.DMXHWOut[485] <-> DMX Channel 449-512/Channel 486
//     PlcTask Outputs/g_ast.DMXHWOut[486] <-> DMX Channel 449-512/Channel 487
//     PlcTask Outputs/g_ast.DMXHWOut[487] <-> DMX Channel 449-512/Channel 488
//     PlcTask Outputs/g_ast.DMXHWOut[488] <-> DMX Channel 449-512/Channel 489
//     PlcTask Outputs/g_ast.DMXHWOut[489] <-> DMX Channel 449-512/Channel 490
//     PlcTask Outputs/g_ast.DMXHWOut[48] <-> DMX Channel 1-64/Channel 49
//     PlcTask Outputs/g_ast.DMXHWOut[490] <-> DMX Channel 449-512/Channel 491
//     PlcTask Outputs/g_ast.DMXHWOut[491] <-> DMX Channel 449-512/Channel 492
//     PlcTask Outputs/g_ast.DMXHWOut[492] <-> DMX Channel 449-512/Channel 493
//     PlcTask Outputs/g_ast.DMXHWOut[493] <-> DMX Channel 449-512/Channel 494
//     PlcTask Outputs/g_ast.DMXHWOut[494] <-> DMX Channel 449-512/Channel 495
//     PlcTask Outputs/g_ast.DMXHWOut[495] <-> DMX Channel 449-512/Channel 496
//     PlcTask Outputs/g_ast.DMXHWOut[496] <-> DMX Channel 449-512/Channel 497
//     PlcTask Outputs/g_ast.DMXHWOut[497] <-> DMX Channel 449-512/Channel 498
//     PlcTask Outputs/g_ast.DMXHWOut[498] <-> DMX Channel 449-512/Channel 499
//     PlcTask Outputs/g_ast.DMXHWOut[499] <-> DMX Channel 449-512/Channel 500
//     PlcTask Outputs/g_ast.DMXHWOut[49] <-> DMX Channel 1-64/Channel 50
//     PlcTask Outputs/g_ast.DMXHWOut[4] <-> DMX Channel 1-64/Channel 5
//     PlcTask Outputs/g_ast.DMXHWOut[500] <-> DMX Channel 449-512/Channel 501
//     PlcTask Outputs/g_ast.DMXHWOut[501] <-> DMX Channel 449-512/Channel 502
//     PlcTask Outputs/g_ast.DMXHWOut[502] <-> DMX Channel 449-512/Channel 503
//     PlcTask Outputs/g_ast.DMXHWOut[503] <-> DMX Channel 449-512/Channel 504
//     PlcTask Outputs/g_ast.DMXHWOut[504] <-> DMX Channel 449-512/Channel 505
//     PlcTask Outputs/g_ast.DMXHWOut[505] <-> DMX Channel 449-512/Channel 506
//     PlcTask Outputs/g_ast.DMXHWOut[506] <-> DMX Channel 449-512/Channel 507
//     PlcTask Outputs/g_ast.DMXHWOut[507] <-> DMX Channel 449-512/Channel 508
//     PlcTask Outputs/g_ast.DMXHWOut[508] <-> DMX Channel 449-512/Channel 509
//     PlcTask Outputs/g_ast.DMXHWOut[509] <-> DMX Channel 449-512/Channel 510
//     PlcTask Outputs/g_ast.DMXHWOut[50] <-> DMX Channel 1-64/Channel 51
//     PlcTask Outputs/g_ast.DMXHWOut[510] <-> DMX Channel 449-512/Channel 511
//     PlcTask Outputs/g_ast.DMXHWOut[511] <-> DMX Channel 449-512/Channel 512
//     PlcTask Outputs/g_ast.DMXHWOut[51] <-> DMX Channel 1-64/Channel 52
//     PlcTask Outputs/g_ast.DMXHWOut[52] <-> DMX Channel 1-64/Channel 53
//     PlcTask Outputs/g_ast.DMXHWOut[53] <-> DMX Channel 1-64/Channel 54
//     PlcTask Outputs/g_ast.DMXHWOut[54] <-> DMX Channel 1-64/Channel 55
//     PlcTask Outputs/g_ast.DMXHWOut[55] <-> DMX Channel 1-64/Channel 56
//     PlcTask Outputs/g_ast.DMXHWOut[56] <-> DMX Channel 1-64/Channel 57
//     PlcTask Outputs/g_ast.DMXHWOut[57] <-> DMX Channel 1-64/Channel 58
//     PlcTask Outputs/g_ast.DMXHWOut[58] <-> DMX Channel 1-64/Channel 59
//     PlcTask Outputs/g_ast.DMXHWOut[59] <-> DMX Channel 1-64/Channel 60
//     PlcTask Outputs/g_ast.DMXHWOut[5] <-> DMX Channel 1-64/Channel 6
//     PlcTask Outputs/g_ast.DMXHWOut[60] <-> DMX Channel 1-64/Channel 61
//     PlcTask Outputs/g_ast.DMXHWOut[61] <-> DMX Channel 1-64/Channel 62
//     PlcTask Outputs/g_ast.DMXHWOut[62] <-> DMX Channel 1-64/Channel 63
//     PlcTask Outputs/g_ast.DMXHWOut[63] <-> DMX Channel 1-64/Channel 64
//     PlcTask Outputs/g_ast.DMXHWOut[64] <-> DMX Channel 65-128/Channel 65
//     PlcTask Outputs/g_ast.DMXHWOut[65] <-> DMX Channel 65-128/Channel 66
//     PlcTask Outputs/g_ast.DMXHWOut[66] <-> DMX Channel 65-128/Channel 67
//     PlcTask Outputs/g_ast.DMXHWOut[67] <-> DMX Channel 65-128/Channel 68
//     PlcTask Outputs/g_ast.DMXHWOut[68] <-> DMX Channel 65-128/Channel 69
//     PlcTask Outputs/g_ast.DMXHWOut[69] <-> DMX Channel 65-128/Channel 70
//     PlcTask Outputs/g_ast.DMXHWOut[6] <-> DMX Channel 1-64/Channel 7
//     PlcTask Outputs/g_ast.DMXHWOut[70] <-> DMX Channel 65-128/Channel 71
//     PlcTask Outputs/g_ast.DMXHWOut[71] <-> DMX Channel 65-128/Channel 72
//     PlcTask Outputs/g_ast.DMXHWOut[72] <-> DMX Channel 65-128/Channel 73
//     PlcTask Outputs/g_ast.DMXHWOut[73] <-> DMX Channel 65-128/Channel 74
//     PlcTask Outputs/g_ast.DMXHWOut[74] <-> DMX Channel 65-128/Channel 75
//     PlcTask Outputs/g_ast.DMXHWOut[75] <-> DMX Channel 65-128/Channel 76
//     PlcTask Outputs/g_ast.DMXHWOut[76] <-> DMX Channel 65-128/Channel 77
//     PlcTask Outputs/g_ast.DMXHWOut[77] <-> DMX Channel 65-128/Channel 78
//     PlcTask Outputs/g_ast.DMXHWOut[78] <-> DMX Channel 65-128/Channel 79
//     PlcTask Outputs/g_ast.DMXHWOut[79] <-> DMX Channel 65-128/Channel 80
//     PlcTask Outputs/g_ast.DMXHWOut[7] <-> DMX Channel 1-64/Channel 8
//     PlcTask Outputs/g_ast.DMXHWOut[80] <-> DMX Channel 65-128/Channel 81
//     PlcTask Outputs/g_ast.DMXHWOut[81] <-> DMX Channel 65-128/Channel 82
//     PlcTask Outputs/g_ast.DMXHWOut[82] <-> DMX Channel 65-128/Channel 83
//     PlcTask Outputs/g_ast.DMXHWOut[83] <-> DMX Channel 65-128/Channel 84
//     PlcTask Outputs/g_ast.DMXHWOut[84] <-> DMX Channel 65-128/Channel 85
//     PlcTask Outputs/g_ast.DMXHWOut[85] <-> DMX Channel 65-128/Channel 86
//     PlcTask Outputs/g_ast.DMXHWOut[86] <-> DMX Channel 65-128/Channel 87
//     PlcTask Outputs/g_ast.DMXHWOut[87] <-> DMX Channel 65-128/Channel 88
//     PlcTask Outputs/g_ast.DMXHWOut[88] <-> DMX Channel 65-128/Channel 89
//     PlcTask Outputs/g_ast.DMXHWOut[89] <-> DMX Channel 65-128/Channel 90
//     PlcTask Outputs/g_ast.DMXHWOut[8] <-> DMX Channel 1-64/Channel 9
//     PlcTask Outputs/g_ast.DMXHWOut[90] <-> DMX Channel 65-128/Channel 91
//     PlcTask Outputs/g_ast.DMXHWOut[91] <-> DMX Channel 65-128/Channel 92
//     PlcTask Outputs/g_ast.DMXHWOut[92] <-> DMX Channel 65-128/Channel 93
//     PlcTask Outputs/g_ast.DMXHWOut[93] <-> DMX Channel 65-128/Channel 94
//     PlcTask Outputs/g_ast.DMXHWOut[94] <-> DMX Channel 65-128/Channel 95
//     PlcTask Outputs/g_ast.DMXHWOut[95] <-> DMX Channel 65-128/Channel 96
//     PlcTask Outputs/g_ast.DMXHWOut[96] <-> DMX Channel 65-128/Channel 97
//     PlcTask Outputs/g_ast.DMXHWOut[97] <-> DMX Channel 65-128/Channel 98
//     PlcTask Outputs/g_ast.DMXHWOut[98] <-> DMX Channel 65-128/Channel 99
//     PlcTask Outputs/g_ast.DMXHWOut[99] <-> DMX Channel 65-128/Channel 100
//     PlcTask Outputs/g_ast.DMXHWOut[9] <-> DMX Channel 1-64/Channel 10
//     PlcTask Outputs/gc.wChannelLength <-> DMX Control/Channel length
//   CSVExample/CSVExample Instance <-> Device 1 (EtherCAT)/Term 1 (EK1100)/Term 29 (EL1008)
//     PlcTask Inputs/g_ast.arrInputPNP[{24..31}] <-> Channel {1..8}/Input  (8 links)
//   CSVExample/CSVExample Instance <-> Device 1 (EtherCAT)/Term 1 (EK1100)/Term 3 (EL1008)
//     PlcTask Inputs/g_ast.arrInputPNP[{0..7}] <-> Channel {1..8}/Input  (8 links)
//   CSVExample/CSVExample Instance <-> Device 1 (EtherCAT)/Term 1 (EK1100)/Term 30 (EL1008)
//     PlcTask Inputs/g_ast.arrInputPNP[{32..39}] <-> Channel {1..8}/Input  (8 links)
//   CSVExample/CSVExample Instance <-> Device 1 (EtherCAT)/Term 1 (EK1100)/Term 31 (EL1008)
//     PlcTask Inputs/g_ast.arrInputPNP[{40..47}] <-> Channel {1..8}/Input  (8 links)
//   CSVExample/CSVExample Instance <-> Device 1 (EtherCAT)/Term 1 (EK1100)/Term 32 (EL1008)
//     PlcTask Inputs/g_ast.arrInputPNP[{48..55}] <-> Channel {1..8}/Input  (8 links)
//   CSVExample/CSVExample Instance <-> Device 1 (EtherCAT)/Term 1 (EK1100)/Term 33 (EL1008)
//     PlcTask Inputs/g_ast.arrInputPNP[{56..63}] <-> Channel {1..8}/Input  (8 links)
//   CSVExample/CSVExample Instance <-> Device 1 (EtherCAT)/Term 1 (EK1100)/Term 34 (EL1008)
//     PlcTask Inputs/g_ast.arrInputPNP[{64..71}] <-> Channel {1..8}/Input  (8 links)
//   CSVExample/CSVExample Instance <-> Device 1 (EtherCAT)/Term 1 (EK1100)/Term 35 (EL1008)
//     PlcTask Inputs/g_ast.arrInputPNP[{72..79}] <-> Channel {1..8}/Input  (8 links)
//   CSVExample/CSVExample Instance <-> Device 1 (EtherCAT)/Term 1 (EK1100)/Term 36 (EL1088)
//     PlcTask Inputs/g_ast.arrInputNPN[{0..7}] <-> Channel {1..8}/Input  (8 links)
//   CSVExample/CSVExample Instance <-> Device 1 (EtherCAT)/Term 1 (EK1100)/Term 37 (EL1088)
//     PlcTask Inputs/g_ast.arrInputNPN[{8..15}] <-> Channel {1..8}/Input  (8 links)
//   CSVExample/CSVExample Instance <-> Device 1 (EtherCAT)/Term 1 (EK1100)/Term 38 (EL1088)
//     PlcTask Inputs/g_ast.arrInputNPN[{16..23}] <-> Channel {1..8}/Input  (8 links)
//   CSVExample/CSVExample Instance <-> Device 1 (EtherCAT)/Term 1 (EK1100)/Term 39 (EL1088)
//     PlcTask Inputs/g_ast.arrInputNPN[{24..31}] <-> Channel {1..8}/Input  (8 links)
//   CSVExample/CSVExample Instance <-> Device 1 (EtherCAT)/Term 1 (EK1100)/Term 4 (EL1008)
//     PlcTask Inputs/g_ast.arrInputPNP[{8..15}] <-> Channel {1..8}/Input  (8 links)
//   CSVExample/CSVExample Instance <-> Device 1 (EtherCAT)/Term 1 (EK1100)/Term 40 (EL1088)
//     PlcTask Inputs/g_ast.arrInputNPN[{32..39}] <-> Channel {1..8}/Input  (8 links)
//   CSVExample/CSVExample Instance <-> Device 1 (EtherCAT)/Term 1 (EK1100)/Term 42 (EL1088)
//     PlcTask Inputs/g_ast.arrInputNPN[{40..47}] <-> Channel {1..8}/Input  (8 links)
//   CSVExample/CSVExample Instance <-> Device 1 (EtherCAT)/Term 1 (EK1100)/Term 43 (EL1088)
//     PlcTask Inputs/g_ast.arrInputNPN[{48..55}] <-> Channel {1..8}/Input  (8 links)
//   CSVExample/CSVExample Instance <-> Device 1 (EtherCAT)/Term 1 (EK1100)/Term 44 (EL1088)
//     PlcTask Inputs/g_ast.arrInputNPN[{56..63}] <-> Channel {1..8}/Input  (8 links)
//   CSVExample/CSVExample Instance <-> Device 1 (EtherCAT)/Term 1 (EK1100)/Term 45 (EL1088)
//     PlcTask Inputs/g_ast.arrInputNPN[{64..71}] <-> Channel {1..8}/Input  (8 links)
//   CSVExample/CSVExample Instance <-> Device 1 (EtherCAT)/Term 1 (EK1100)/Term 46 (EL1088)
//     PlcTask Inputs/g_ast.arrInputNPN[{72..79}] <-> Channel {1..8}/Input  (8 links)
//   CSVExample/CSVExample Instance <-> Device 1 (EtherCAT)/Term 1 (EK1100)/Term 5 (EL1008)
//     PlcTask Inputs/g_ast.arrInputPNP[{16..23}] <-> Channel {1..8}/Input  (8 links)

CONFIGURATION CSVExample
    RESOURCE PLC ON TwinCAT3
        TASK PlcTask(INTERVAL := T#10ms, PRIORITY := 20);
        PROGRAM MAIN WITH PlcTask : MAIN;
        PROGRAM DMXTest WITH PlcTask : DMXTest;
        PROGRAM P_TextModeRead WITH PlcTask : P_TextModeRead;
        PROGRAM InterfaceLink WITH PlcTask : InterfaceLink;
        PROGRAM IOParams WITH PlcTask : IOParams;
    END_RESOURCE
END_CONFIGURATION

// ---- DUTs/ENUM_BufferMgmt.TcDUT
{attribute 'qualified_only'}
{attribute 'strict'}
TYPE ENUM_BufferMgmt :
(
	EN_Idle 		:= 0,
	EN_TestWrite	:= 1,
	EN_Test			:= 2,
	EN_Write		:= 3,
	EN_TestWritten	:= 4	
);
END_TYPE

// ---- DUTs/ENUM_SeqSM.TcDUT
{attribute 'qualified_only'}
{attribute 'strict'}
TYPE ENUM_SeqSM :
(
	Once		:=0, //(Lights, Dry Contacts)
	OnceDC		:=1, // Dry Contact (HVAC)
	Twice		:=2 //(Motors)
);
END_TYPE

// ---- DUTs/typ_FB_Debounce/typFBDInput.TcDUT
TYPE typFBDInput :
	STRUCT
		tOnDelay	: TIME;
		tOffDelay	: TIME;
	END_STRUCT
END_TYPE

// ---- DUTs/typ_FB_Debounce/typ_FBInt_Debounce.TcDUT
TYPE typ_FBInt_Debounce :
STRUCT
	I		: typFBDInput;
	IQ		: typFBDInOut;
	Q		: typFBDOutput;
END_STRUCT
END_TYPE

// ---- DUTs/typ_FB_DMX/ENUM_I_Waveform.TcDUT
{attribute 'qualified_only'}
{attribute 'strict'}
TYPE ENUM_I_Waveform :
(
	EN_Square		:= 10,
	EN_Rand			:= 20,
	EN_Sin			:= 30,
	EN_Triangle		:= 40,
	EN_SubTriFall	:= 42,
	EN_SubTriRise	:= 44, 
	EN_Saw			:= 50,
	EN_Ramp			:= 60,
	EN_GateConfig	:= 70, //Non-periodic Square
	EN_GateCtrl		:= 80 //Non-periodic Square
);
END_TYPE

// ---- DUTs/typ_FB_DMX/typDMXInput.TcDUT
TYPE typDMXInput :
STRUCT
	ENWaveform		: ENUM_I_Waveform;
	ENValRange		: ENUM_I_ValRange;
	fDutyCycle		: REAL; // just for Square Wave;
	fFrequency		: REAL;  // Frequency of cycling, expressed in Hz
	fOffset			: REAL; // 0-100% mapped to 8-bit (by Map Function)
	fLevel			: REAL; // 0-100% mapped to 8-bit (by Map Function)
	usiBitDepth		: USINT; // 1-8
	fPhase			: REAL; // 0-100% mapped to 8-bit (by Map Function)
	fDelay			: REAL; // 0-100% mapped to 8-bit (by Map Function)
	usiDelayDiv		: USINT; // to Delay the step of the Delay Divisor; for example, '2' would delay every second pulse by the amount spec'd by fDelay
	usiInputConfig	: USINT; // BYTE Value specified in USINT [0-255]
END_STRUCT
END_TYPE

// ---- DUTs/typ_FB_DMX/typDMXOutput.TcDUT
TYPE typDMXOutput :
STRUCT
	byStatValue			: BYTE;
	fFnGeneratorVal		: LREAL;
END_STRUCT
END_TYPE

// ---- DUTs/typ_FB_DMX/typ_FBInt_DMX.TcDUT
TYPE typ_FBInt_DMX :
STRUCT
	I		: typDMXInput;
	IQ		: typDMXInOut;
	Q		: typDMXOutput;
END_STRUCT
END_TYPE

// ---- GVLs/gc.TcGVL
{attribute 'qualified_only'}
VAR_GLOBAL CONSTANT
	uiMaxNrOfDMXChannel				: UINT := 511;
	wChannelLength			AT %Q*	: WORD := 512;
	fPi								: REAL	:= 3.141592653589793238462643383279;
	uiMinNrDMXTestCh				: UINT	:= 0;
	uiMaxNrDMXTestCh				: UINT	:= 79; // Dictated by hardware constraints (80 channels input)
	uiChannelsUT	 				: UINT	:= 80;		(*Channels Under Test *)
	uiVisualizationIndexLim			: UINT	:= 7;
	uiDUTConfigCountSplit			: UINT	:= 255;
	uiChannelSplitCount				: UINT	:= 256;
END_VAR

// ---- GVLs/gFB.TcGVL
{attribute 'qualified_only'}
VAR_GLOBAL
	arrFB_DMX				: ARRAY[0..gc.uiMaxNrOfDMXChannel] OF FB_DMX;
	arrFB_DebouncePNP		: ARRAY[0..gc.uiMaxNrDMXTestCh] OF FB_InputDebounce;
	arrFB_DebounceNPN		: ARRAY[0..gc.uiMaxNrDMXTestCh] OF FB_InputDebounce;
END_VAR

// ---- GVLs/GVL.TcGVL
VAR_GLOBAL CONSTANT
	MAX_CSV_ROWS 			: UDINT := 512; (*gc.uiMaxNrOfDMXChannel*)
	MAX_CSV_COLUMNS 		: UDINT := 2;
	MAX_CSV_FIELD_LENGTH	: UDINT := 4;
END_VAR

// ---- GVLs/g_ast.TcGVL
{attribute 'qualified_only'}
VAR_GLOBAL
		// INPUT array structs for mapping to Physical I/O (PIO)
//	gast_SensorInput		AT %I* : ARRAY[0..gc.usiMaxNrOfSensor] OF typ_FBInt_Debounce;
	
	//2 Sensors on each valve (assumed)
//	gast_ValveSensorInput	AT %I* : ARRAY[0..(2*gc.usiMaxNrOfValveCtrl)] OF typ_FBInt_Debounce;
//	gast_AnalogInput		AT %I* : ARRAY[0..gc.usiMaxNrOfAnalogIn] OF typ_FBInt_Analog;
	
// OUTPUT array structs for mapping to Physical I/O (PIO)
//	gast_ValveCtrlOutput	AT %Q* : ARRAY[0..gc.usiMaxNrOfValveCtrl] OF typ_FBInt_ValveCtrl;
//	gast_DigCtrlOutput		AT %Q* : ARRAY[0..gc.usiMaxNrOfDigCtrl] OF typ_FBInt_DigCtrl;
	DMX						: ARRAY[0..gc.uiMaxNrOfDMXChannel] OF typ_FBInt_DMX;
	DMXPhysOut				: ARRAY[0..gc.uiMaxNrOfDMXChannel] OF BYTE; (* software buffer *)
	DMXHWOut		AT %Q*	: ARRAY[0..gc.uiMaxNrOfDMXChannel] OF BYTE; (* Defined to allow Multi-Link of I/O in Physical I/O tree *)
	arrFBIntPNP				: ARRAY[0..gc.uiMaxNrDMXTestCh] OF typ_FBInt_Debounce;
	arrFBIntNPN				: ARRAY[0..gc.uiMaxNrDMXTestCh] OF typ_FBInt_Debounce;
	arrInputPNP		AT %I*	: ARRAY[0..gc.uiMaxNrDMXTestCh] OF BOOL;
	arrInputNPN		AT %I*	: ARRAY[0..gc.uiMaxNrDMXTestCh] OF BOOL;
END_VAR

// ---- POUs/MAIN.TcPOU
PROGRAM MAIN
VAR
(*	In USA/UK the CSV field separator is a comma.
	In Germany and some other European countries the CSV field separator is a semicolon. *)
	bChangeSeparatorToComma	: BOOL := TRUE;
	iLoopDMXCtrlQ			: INT;
	ENBufferMgmt			: ENUM_BufferMgmt;
	diMapTest				: DINT;
	arrfFnGenerVal			: ARRAY[0..gc.uiMaxNrOfDMXChannel] OF LREAL;
	uiIndexFnGenSend		: UINT;
	uiIndexFnGenRtn			: UINT;
	uiLoopDebouncePNPII		: UINT;
	uiLoopDebounceNPNII		: UINT;
END_VAR

IF bChangeSeparatorToComma THEN
	DEFAULT_CSV_FIELD_SEP := 16#2C;(* Comma ASCII code *)
ELSE
	DEFAULT_CSV_FIELD_SEP := 16#3B;(* Semicolon ASCII code *)
END_IF

P_TextModeRead();(* This sample program opens and reads CSV file in text mode *)

P_TextModeWrite();(* This sample program opens and writes CSV file in text mode *)

P_BinaryModeRead();(* This sample program opens and reads CSV file in binary mode *)

P_BinaryModeWrite();(* This sample program opens and writes CSV file in binary mode *)

P_ArgToConvExample();(* This sample program shows the usage of the ARG_TO_CSVFIELD and CSVFILED_TO_ARG conversion functions *)

P_StringToConvExample();(* This sample program shows the usage of the STRING_TO_CSVFIELD and CSVFIELD_TO_STRING conversion functions *)

//DMX Code
//Special case to handle function calls outside ("send" and "return" to FB for SIN (or potentially other) function output types)
IF g_ast.DMX[uiIndexFnGenSend].I.ENWaveform = ENUM_I_Waveform.EN_Sin THEN
	FOR uiIndexFnGenSend := 0 TO gc.uiMaxNrOfDMXChannel BY 1 DO
		//SIN Function MUST be called from MAIN; not within FunctionBlock (FB_DMX)
		arrfFnGenerVal[uiIndexFnGenSend]	:= 1+(SIN(g_ast.DMX[uiIndexFnGenSend].IQ.fFnGenerValTempSin));
	END_FOR
	
	FOR uiIndexFnGenRtn := 0 TO gc.uiMaxNrOfDMXChannel BY 1 DO
		//SIN Function MUST be called from MAIN; not within FunctionBlock (FB_DMX)
		g_ast.DMX[uiIndexFnGenRtn].IQ.fFnGenerValRtn	:= arrfFnGenerVal[uiIndexFnGenRtn];
	END_FOR
END_IF

//Link AST to hardware inputs - PNP
FOR uiLoopDebouncePNPII	:= 0 TO gc.uiMaxNrDMXTestCh BY 1 DO
	g_ast.arrFBIntPNP[uiLoopDebouncePNPII].IQ.xTrig		:= g_ast.arrInputPNP[uiLoopDebouncePNPII];
END_FOR

//Link AST to hardware inputs - NPN
FOR uiLoopDebounceNPNII	:= 0 TO gc.uiMaxNrDMXTestCh BY 1 DO
	g_ast.arrFBIntNPN[uiLoopDebounceNPNII].IQ.xTrig		:= g_ast.arrInputNPN[uiLoopDebounceNPNII];
END_FOR

END_PROGRAM

// ---- POUs/CSV read_write in binary mode/P_BinaryModeRead.TcPOU
(* Reading of CSV file in binary mode. Field values may contain non-printing control characters (binary data or special characters like line feed, carriage return or quotation mark...). *)
PROGRAM P_BinaryModeRead
VAR
	bRead		: BOOL := FALSE;(* Rising edge starts program execution *)
	sNetId		: T_AmsNetId := '';	(* TwinCAT system network address *)
	sFileName	: T_MaxString := 'C:\Temp\BinaryModeGen.csv';(* CSV source file path and name *)
	bBusy		: BOOL;
	bError		: BOOL;
	nErrId		: UDINT;
	nRow	 	: UDINT 	:= 0;(* Row number (record) *)
	nColumn		: UDINT 	:= 0;(* Column number (record field) *)
	cbDone		: UDINT 	:= 0;(* Counts allready parsed data bytes *)
	hFile		: UINT		:= 0;(* File handle of the source file *)
	step		: DWORD 	:= 0;
	fbFileOpen	: FB_FileOpen;(* Opens file *)
	fbFileClose	: FB_FileClose;(* Closes file *)
	fbFileRead	: FB_FileRead;(* Writes binary data *)
	fbReader	: FB_CSVMemBufferReader;(* Helper function block used to parse CSV data bytes *)

	record		: ARRAY[0..1024] OF BYTE;(* Binary row data buffer. The size of this buffer have to be > length of longest record line + 2 (CRLF)  *)
	cbRecord	: UDINT := 0;(* Number of bytes in row buffer *)
	cbField		: UDINT;(* Number of bytes in field buffer *)

	database	: ARRAY[0..MAX_CSV_ROWS ] OF ST_CSV_Record;(* Target PLC database *)
END_VAR

CASE step OF
	0:	(* Wait for rising edge at bRead variable *)
		IF bRead THEN
			bRead 	:= FALSE;
			bBusy 	:= TRUE;
			bError	:= FALSE;
			nErrId	:= 0;
			hFile	:= 0;
			nRow	:= 0;
			nColumn	:= 0;
			cbRecord:= 0;
			cbDone 	:= 0;
			step 	:= 1;
		END_IF

	1:	(* Open source file *)
		fbFileOpen(  bExecute := FALSE  );
		fbFileOpen( sNetId := sNetId, sPathName := sFileName, nMode := FOPEN_MODEREAD OR FOPEN_MODEBINARY,(* Open file in BINARY mode! *)
					ePath := PATH_GENERIC, bExecute := TRUE );
		step := 2;

	2:(* Wait until open not busy *)
		fbFileOpen( bExecute := FALSE, bError => bError, nErrID => nErrID, hFile => hFile );
		IF NOT fbFileOpen.bBusy THEN
			IF NOT fbFileOpen.bError THEN
				step := 3;
			ELSE(* Error: file not found? *)
				step := 100;
			END_IF
		END_IF

	3:	(* Read data bytes from file *)
		fbFileRead( bExecute := FALSE );
		fbFileRead( sNetId := sNetId, hFile := hFile, pReadBuff := ADR( record[ cbRecord ] ), cbReadLen := SIZEOF( record ) - cbRecord, bExecute :=TRUE );
		step := 4;

	4:(* Wait until read not busy *)
		fbFileRead( bExecute := FALSE, bError => bError, nErrID => nErrID );
		IF NOT fbFileRead.bBusy THEN
			IF NOT fbFileRead.bError THEN
				IF fbFileRead.bEOF THEN
					step := 10;(* End of file reached => Close source file *)
				ELSE
					cbRecord := cbRecord + fbFileRead.cbRead;(* Recalculate the new size of data buffer *)
					step := 5;(* Parse binary data *)
				END_IF
			ELSE(* Error *)
				step := 100;
			END_IF
		END_IF

	5:(* Parse binary data *)
		cbDone := 0;(* Reset number of parsed data bytes *)
		fbReader.eCmd := eEnumCmd_First;(* Read first field value *)
		REPEAT
			fbReader( pBuffer := ADR( record ), cbBuffer := cbRecord );
			IF fbReader.bOk THEN
				fbReader.eCmd := eEnumCmd_Next;(* Read next field value *)
				cbDone := cbDone + fbReader.cbRead;(* Count the number of successfully parsed data bytes *)

				IF ( nRow <= MAX_CSV_ROWS ) THEN
					(* Convert every CSV data field to PLC data field format *)
					CASE nColumn OF
						0:(* sName : T_MaxString *)
							cbField := CSVFIELD_TO_ARG( fbReader.pValue, fbReader.cbValue,  TRUE, F_STRING( database[nRow].sName ) );
						1:(* nNumber : UDINT *)
							cbField := CSVFIELD_TO_ARG( fbReader.pValue, fbReader.cbValue,  TRUE, F_UDINT( database[nRow].nNumber ) );
						2:(* fPos : LREAL *)
							cbField := CSVFIELD_TO_ARG( fbReader.pValue, fbReader.cbValue,  TRUE, F_LREAL( database[nRow].fPos ) );
						3:(* bOP : BOOL *)
							cbField := CSVFIELD_TO_ARG( fbReader.pValue, fbReader.cbValue,  TRUE, F_BOOL( database[nRow].bOP ) );
						4:(* sDesc : STRING(40) *)
							cbField := CSVFIELD_TO_ARG( fbReader.pValue, fbReader.cbValue,  TRUE, F_BIGTYPE( ADR( database[nRow].sDesc ), SIZEOF( database[nRow].sDesc ) ) );
						5:(* data : ARRAY[0..7] OF BYTE *)
							cbField := CSVFIELD_TO_ARG( fbReader.pValue, fbReader.cbValue,  TRUE, F_BIGTYPE( ADR( database[nRow].data ), SIZEOF( database[nRow].data ) ) );
					ELSE
						;
					END_CASE
				END_IF

				nColumn := nColumn + 1;(* Increment number of read columns *)
				IF fbReader.bCRLF THEN(* CRLF == TRUE => End of reacord reached *)
					nRow 		:= nRow + 1;(* Increment number of read records *)
					nColumn 	:= 0;(* Reset number of columns *)
				END_IF

			ELSE(* Error: End of buffer reached or all fields parsed *)
				cbRecord := MEMMOVE( ADR( record ), ADR( record[ cbDone ] ), cbRecord - cbDone );(* Shift left the remaining (not allready read) data bytes *)
				step := 3;(* Read new data bytes *)
			END_IF
		UNTIL NOT fbReader.bOk
		END_REPEAT

	10:	(* Close source file *)
		fbFileClose( bExecute := FALSE );
		fbFileClose( sNetId := sNetId, hFile := hFile, bExecute := TRUE );
		step := 11;

	11:(* Wait until close not busy *)
		fbFileClose( bExecute := FALSE, bError => bError, nErrID => nErrID );
		IF ( NOT fbFileClose.bBusy ) THEN
			hFile := 0;
			step := 100;
		END_IF

	100: (* Error or ready step => cleanup *)
		IF ( hFile <> 0 ) THEN
			step := 10; (* Close the source file *)
		ELSE
			bBusy := FALSE;
			step := 0;	(* Ready *)
		END_IF

END_CASE

END_PROGRAM

// ---- POUs/P_ArgToConvExample.TcPOU
PROGRAM P_ArgToConvExample
VAR
	(* PLC data to be converted to or from CSV format *)
	bOperating	: BOOL := TRUE;
	fAxPos		: LREAL := 12.2;
	nCounter 	: UDINT := 7;
	sName		: T_MaxString := 'Module: "XAF", $04$05, 20';
	binData		: ARRAY[0..9] OF BYTE :=[ 0, 1, 2, 3, 4, 5, 6, 7, 8, 9];
	sShort		: STRING(10) := 'XAF';

	(* conversion buffer *)
	field1 : ARRAY[0..50 ] OF BYTE;
	field2 : ARRAY[0..50 ] OF BYTE;
	field3 : ARRAY[0..50 ] OF BYTE;
	field4 : ARRAY[0..50 ] OF BYTE;
	field5 : ARRAY[0..50 ] OF BYTE;
	field6 : ARRAY[0..50 ] OF BYTE;

	cbField1 : UDINT;
	cbField2 : UDINT;
	cbField3 : UDINT;
	cbField4 : UDINT;
	cbField5 : UDINT;
	cbField6 : UDINT;

	cbVar1 : UDINT;
	cbVar2 : UDINT;
	cbVar3 : UDINT;
	cbVar4 : UDINT;
	cbVar5 : UDINT;
	cbVar6 : UDINT;

END_VAR

cbField1 := ARG_TO_CSVFIELD( F_BOOL( bOperating ), TRUE, ADR( field1 ), SIZEOF( field1 ) );
cbField2 := ARG_TO_CSVFIELD( F_LREAL( fAxPos ), TRUE, ADR( field2 ), SIZEOF( field2 ) );
cbField3 := ARG_TO_CSVFIELD( F_UDINT( nCounter ), TRUE, ADR( field3 ), SIZEOF( field3 ) );
cbField4 := ARG_TO_CSVFIELD( F_STRING( sName ), TRUE, ADR( field4 ), SIZEOF( field4 ) );
cbField5 := ARG_TO_CSVFIELD( F_BIGTYPE( ADR( binData ), SIZEOF( binData ) ), TRUE, ADR( field5 ), SIZEOF( field5 ) );
cbField6 := ARG_TO_CSVFIELD( F_BIGTYPE( ADR( sShort ), INT_TO_DWORD( LEN( sShort ) ) ), TRUE, ADR( field6 ), SIZEOF( field6 ) );

cbVar1 := CSVFIELD_TO_ARG( ADR( field1 ), cbField1, TRUE, F_BOOL( bOperating ) );
cbVar2 := CSVFIELD_TO_ARG( ADR( field2 ), cbField2, TRUE, F_LREAL( fAxPos ) );
cbVar3 := CSVFIELD_TO_ARG( ADR( field3 ), cbField3, TRUE, F_UDINT( nCounter ) );
cbVar4 := CSVFIELD_TO_ARG( ADR( field4 ), cbField4, TRUE, F_STRING( sName ) );
cbVar5 := CSVFIELD_TO_ARG( ADR( field5 ), cbField5, TRUE, F_BIGTYPE( ADR( binData ), SIZEOF( binData ) ) );
cbVar6 := CSVFIELD_TO_ARG( ADR( field6 ), cbField6, TRUE, F_BIGTYPE( ADR( sShort ), INT_TO_DWORD( LEN( sShort ) ) ) );

END_PROGRAM

// ---- POUs/P_StringToConvExample.TcPOU
PROGRAM P_StringToConvExample
VAR
	s1	: STRING;
	s2	: STRING;
END_VAR

s1 := STRING_TO_CSVFIELD( 'Module_"ALFA_$05"_6', TRUE  );
s2 := STRING_TO_CSVFIELD( 'Module_50', FALSE );

s1 := CSVFIELD_TO_STRING( '"ab_$04_$05_cd-""ALFA""_5"', TRUE  );
s2 := CSVFIELD_TO_STRING( 'Module_50', FALSE );

END_PROGRAM

// ---- POUs/DMXTest.TcPOU
PROGRAM DMXTest
VAR
	xConfigSet					: BOOL;
	xStatTestInProgress			: BOOL;
	xDMXSeqTestInProgressOnce	: BOOL;
	xDMXSeqTestInProgressTwice	: BOOL;
	xDMXSeqTestInProgressOnceDC	: BOOL;
	uiCounter2					: UINT;
	uiCounter3					: UINT;
	uiCounter4					: UINT;
	uiCounter5					: UINT;
	uiCounter6					: UINT;
	uiCounter7					: UINT;
	uiCounter8					: UINT;
	uiCounter9					: UINT;
	uiDedicatedRcvdRTIndex		: UINT;
	uiContinuousRTIndex			: UINT;
	
	uiForLoopCfgIndex			: UINT;
//	uiForLoopCtrlWriteIndex		: UINT;
//	uiForLoopCtrlWriteIndex2	: UINT;	
	uiLoopExpctdIndex			: UINT;
	uiForLoopClearExpctd		: UINT;
	uiLoopRcvIndex				: UINT;
	uiByteIndex					: UINT;
	iForLoopRecipeFindMin		: INT;
	iForLoopRecipeFindMax		: INT;
	iForLoopRecipeFindMax1		: INT;
	iForLoopRecipeMin			: INT;
	uiForLoopRecipe				: UINT;
	uiLoopIterDMXDUTArraySeq	: UINT;
	uiLoopIterDMXDUTArrayM		: UINT;
	uiLoopIterDUTArray24V		: UINT;
	uiLoopIterDUTArrayGND		: UINT;
	uiLoopIterTestArrSeq		: UINT;
	uiLoopIterTestArrM			: UINT;
	uiLoopIterTestArr24V		: UINT;
	uiLoopIterTestArrGND		: UINT;	
	iCompareStaticSM			: INT;
	iCompareSeq					: ARRAY[0..ENUM_SeqSM.Twice] OF INT;
	iParseFile					: INT;
	iSetConfig					: INT;
	iSetExpctdBufferSM			: INT;
	iReindexExpctedBufferSM		: INT;
	rt_RunStaticTest			: R_TRIG;
	rt_RunSeqTestOnce			: R_TRIG;
	rt_RunSeqTestOnceDC			: R_TRIG;
	rt_RunSeqTestTwice			: R_TRIG;
	rt_ResetTest				: R_TRIG;
	rt_ResetTestSeq				: R_TRIG;
	rt_ResetTestSeqDC			: R_TRIG;
	r_tStaticTestDone			: R_TRIG;
	
	//Arrays (Refactor 30-09-21)
	arr_uiRecipeIndexTmp		: ARRAY[0..gc.uiDUTConfigCountSplit] OF UINT;
 	arruiDMXChDUTTmp			: ARRAY[0..gc.uiDUTConfigCountSplit] OF UINT;
	arrsDUTChTypeTmp			: ARRAY[0..gc.uiDUTConfigCountSplit] OF STRING[3];	
	arr_uiRecipeIndex			: ARRAY[0..gc.uiDUTConfigCountSplit] OF UINT;
 	arruiDMXChDUT				: ARRAY[0..gc.uiDUTConfigCountSplit] OF UINT;
	arrsDUTChType				: ARRAY[0..gc.uiDUTConfigCountSplit] OF STRING[3];
	xFileImported				: BOOL;
	arr_usiRecipeSettingTmp		: ARRAY[0..gc.uiMaxNrOfDMXChannel] OF USINT;
	arr_usiRecipeSetting		: ARRAY[0..gc.uiMaxNrOfDMXChannel] OF USINT;






	
		
	arrxRcvdBufferPNP24V		: ARRAY[0..gc.uiMaxNrDMXTestCh] OF BOOL;
	arrxRcvdBufferNPN24V		: ARRAY[0..gc.uiMaxNrDMXTestCh] OF BOOL;
	arrxRcvdBufferPNPGND		: ARRAY[0..gc.uiMaxNrDMXTestCh] OF BOOL;
	arrxRcvdBufferNPNGND		: ARRAY[0..gc.uiMaxNrDMXTestCh] OF BOOL;
	
	arrxRcvdBufferPNPSeq		: ARRAY[0..gc.uiMaxNrDMXTestCh] OF BOOL;
	arrxRcvdBufferNPNSeq		: ARRAY[0..gc.uiMaxNrDMXTestCh] OF BOOL;	
	arrxRcvdBufferPNPMotor		: ARRAY[0..gc.uiMaxNrDMXTestCh] OF BOOL;
	arrxRcvdBufferNPNMotor		: ARRAY[0..gc.uiMaxNrDMXTestCh] OF BOOL;
	
	arrxExpctdPNP				: ARRAY[0..gc.uiMaxNrOfDMXChannel] OF BOOL; //What is expected based on the recipe file
	arrxExpctdNPN				: ARRAY[0..gc.uiMaxNrOfDMXChannel] OF BOOL; //What is expected based on the recipe file
	arrxExpctdTmpPNP			: ARRAY[0..gc.uiMaxNrOfDMXChannel] OF BOOL; //What is expected based on the recipe file, reindexed from DUT (usually 0)
	arrxExpctdTmpNPN			: ARRAY[0..gc.uiMaxNrOfDMXChannel] OF BOOL; //What is expected based on the recipe file, reindexed from DUT (usually 0)
	arrxExpctdTmpPNP24V			: ARRAY[0..gc.uiMaxNrDMXTestCh] OF BOOL; //What is expected based on the recipe file, reindexed from DUT (usually 0)
	arrxExpctdTmpNPN24V			: ARRAY[0..gc.uiMaxNrDMXTestCh] OF BOOL; //What is expected based on the recipe file, reindexed from DUT (usually 0)
	arrxExpctdTmpPNPGND			: ARRAY[0..gc.uiMaxNrDMXTestCh] OF BOOL; //What is expected based on the recipe file, reindexed from DUT (usually 0)
	arrxExpctdTmpNPNGND			: ARRAY[0..gc.uiMaxNrDMXTestCh] OF BOOL; //What is expected based on the recipe file, reindexed from DUT (usually 0)

	arrxExpctdTmpPNPSeqDMX		: ARRAY[0..gc.uiMaxNrDMXTestCh] OF BOOL; //What is expected based on the recipe file, reindexed from DUT (usually 0)
	arrxExpctdTmpNPNSeqDMX		: ARRAY[0..gc.uiMaxNrDMXTestCh] OF BOOL; //What is expected based on the recipe file, reindexed from DUT (usually 0)
	arrxExpctdTmpPNPSeqDC		: ARRAY[0..gc.uiMaxNrDMXTestCh] OF BOOL; //What is expected based on the recipe file, reindexed from DUT (usually 0)
	arrxExpctdTmpNPNSeqDC		: ARRAY[0..gc.uiMaxNrDMXTestCh] OF BOOL; //What is expected based on the recipe file, reindexed from DUT (usually 0)

	arrxExpctdTmpPNPSeq			: ARRAY[0..gc.uiMaxNrOfDMXChannel] OF BOOL; //What is expected based on the recipe file, reindexed from DUT (usually 0)
	arrxExpctdTmpNPNSeq			: ARRAY[0..gc.uiMaxNrOfDMXChannel] OF BOOL; //What is expected based on the recipe file, reindexed from DUT (usually 0)
	arrxExpctdTmpPNPMotor		: ARRAY[0..gc.uiMaxNrOfDMXChannel] OF BOOL; //What is expected based on the recipe file, reindexed from DUT (usually 0)
	arrxExpctdTmpNPNMotor		: ARRAY[0..gc.uiMaxNrOfDMXChannel] OF BOOL; //What is expected based on the recipe file, reindexed from DUT (usually 0)
	
	arrxExpctdMaskPNPSeq		: ARRAY[0..gc.uiMaxNrOfDMXChannel] OF BOOL; //Copy the contents of hardware buffer 
	arrxExpctdMaskNPNSeq		: ARRAY[0..gc.uiMaxNrOfDMXChannel] OF BOOL; //Copy the contents of hardware buffer 
	arr_diTestStaticPNP24V		: ARRAY[0..gc.uiMaxNrDMXTestCh] OF DINT;
	arr_diTestStaticNPN24V		: ARRAY[0..gc.uiMaxNrDMXTestCh] OF DINT;
	arr_diTestStaticPNPGND		: ARRAY[0..gc.uiMaxNrDMXTestCh] OF DINT;
	arr_diTestStaticNPNGND		: ARRAY[0..gc.uiMaxNrDMXTestCh] OF DINT;
	arr_diTestPNPSeqOnceLine			: ARRAY[0..gc.uiMaxNrDMXTestCh] OF DINT;
	arr_diTestPNPSeqOnceLineTmp			: ARRAY[0..gc.uiMaxNrDMXTestCh] OF DINT;
	arr_diTestNPNSeqOnceLine			: ARRAY[0..gc.uiMaxNrDMXTestCh] OF DINT;
	arr_diTestNPNSeqOnceLineTmp			: ARRAY[0..gc.uiMaxNrDMXTestCh] OF DINT;

	arr_udiMEMCPYPNPSeqOnceRcvdTmp		: ARRAY[0..gc.uiMaxNrDMXTestCh] OF UDINT;
	arr_udiMEMCPYNPNSeqOnceRcvdTmp		: ARRAY[0..gc.uiMaxNrDMXTestCh] OF UDINT;
			
	diTestStaticPNP24V				: DINT;
	diTestStaticNPN24V				: DINT;
	diTestStaticPNPGND				: DINT;	
	diTestStaticNPNGND				: DINT;
	
	diTestPNPSeqOnceComplete		: DINT;

	arrdiTestPNPSeqOnceComplete		: ARRAY[0..gc.uiMaxNrDMXTestCh] OF DINT;
	arrdiTestPNPSeqOnceCompleteTmp	: ARRAY[0..gc.uiMaxNrDMXTestCh] OF DINT;

	arrdiTestNPNSeqOnceComplete		: ARRAY[0..gc.uiMaxNrDMXTestCh] OF DINT;
	arrdiTestNPNSeqOnceCompleteTmp	: ARRAY[0..gc.uiMaxNrDMXTestCh] OF DINT;

	arrdiTestNPNSeqOnceCompleteProblemIndex		: ARRAY[0..gc.uiMaxNrDMXTestCh] OF DINT;
	
	arrudiStaticCopyResultPNP24V	: ARRAY[0..gc.uiMaxNrOfDMXChannel] OF UDINT;
	arrudiStaticCopyResultNPN24V	: ARRAY[0..gc.uiMaxNrOfDMXChannel] OF UDINT;
	arrudiStaticCopyResultPNPGND	: ARRAY[0..gc.uiMaxNrOfDMXChannel] OF UDINT;
	arrudiStaticCopyResultNPNGND	: ARRAY[0..gc.uiMaxNrOfDMXChannel] OF UDINT;	

	arr_diTestPNPMotorDir1		: ARRAY[0..gc.uiMaxNrDMXTestCh] OF DINT;
	arr_diTestNPNMotorDir1		: ARRAY[0..gc.uiMaxNrDMXTestCh] OF DINT;
	arr_diTestPNPMotorDir2		: ARRAY[0..gc.uiMaxNrDMXTestCh] OF DINT;
	arr_diTestNPNMotorDir2		: ARRAY[0..gc.uiMaxNrDMXTestCh] OF DINT;

	
	
	diCompTestResult			: DINT;
	diCompTestResultTemp		: DINT;
	diTestResultStaticPNP		: DINT;
	diTestResultStaticNPN		: DINT;	

	arrVisu_diTestResult		: ARRAY[0..gc.uiMaxNrDMXTestCh] OF DINT;
	uiVisuIndex					: UINT;
	tonReadWait					: TON;
	tonConvert					: TON;
	tonWriteCopyWait			: TON;
	tonTestIterGap				: TON;
	tTestTime					: TIME;
	tWriteWaitTime				: TIME;
	r_tSetConfig				: R_TRIG;
	uiRecipeIndexRcv			: UINT;
	uiMinRecipeIndex			: UINT;
	uiMaxRecipeIndex			: UINT;
	cuiMinDUTIndex				: UINT	:= 0; // Constant
	uiMaxRecipeIndexTemp		: UINT;
	arruiMotorTestIndices		: ARRAY[0..gc.uiMaxNrOfDMXChannel] OF UINT;
	arruiMotorTestIndicesTmp	: ARRAY[0..gc.uiMaxNrOfDMXChannel] OF UINT;
	arruiSeqTestIndices			: ARRAY[0..gc.uiMaxNrOfDMXChannel] OF UINT;
	arruiSeqTestIndicesTmp		: ARRAY[0..gc.uiMaxNrOfDMXChannel] OF UINT;
	
	arruiSeqTestIndicesDMX			: ARRAY[0..gc.uiMaxNrDMXTestCh] OF UINT;
	arruiSeqTestIndicesDMXSW		: ARRAY[0..gc.uiMaxNrDMXTestCh] OF UINT;
	arruiSeqTestIndicesDMXTmp		: ARRAY[0..gc.uiMaxNrDMXTestCh] OF UINT;
	
	arruiSeqTestIndicesDC			: ARRAY[0..gc.uiMaxNrDMXTestCh] OF UINT;
	arruiSeqTestIndicesDCTmp		: ARRAY[0..gc.uiMaxNrDMXTestCh] OF UINT;	
	
	arrui24VTestIndices			: ARRAY[0..gc.uiMaxNrOfDMXChannel] OF UINT;
	arrui24VTestIndicesTmp		: ARRAY[0..gc.uiMaxNrOfDMXChannel] OF UINT;
	arruiGNDTestIndices			: ARRAY[0..gc.uiMaxNrOfDMXChannel] OF UINT;
	arruiGNDTestIndicesTmp		: ARRAY[0..gc.uiMaxNrOfDMXChannel] OF UINT;
	udiMemCpyResultPNP			: UDINT;
	udiMemCpyResultDMX			: UDINT;	
	r_tSetExpectedBuff			: R_TRIG;
	r_tExpectedBufferSet		: R_TRIG;
	uiLoopExpctdIndexRead		: UINT;
	uiLoopExpctdIndexWrite		: UINT;
	xTestBoolDelete				: BOOL;
	uiForLoopZeroStorageArray	: UINT;
	
	//For DUT Config
	r_tSetDUTVal				: R_TRIG;
	usiDUTVal					: USINT;
	uiForLoopDUTIter			: UINT;
	iSetDUTSM					: INT;
	
	//For 'Invert Recipe Settings'
	uiStartingIndex				: UINT;
	uiEndingIndex				: UINT;
	uiRecipeInvertIter			: UINT;
	R_TInvertRecipe				: R_TRIG;
	iInvertRecipeSM				: INT;
END_VAR

SeqTestOnce();
//SeqTestTwice();
//SeqTestOnceDC();
InvertRecipeSettings();
rt_RunStaticTest();
rt_ResetTest();
r_tSetConfig();//Set config when file is loaded; this condition happens when End-of-File (EOF) is reached; set by HMI button
r_tSetExpectedBuff(CLK:=r_tSetConfig.Q);
r_tExpectedBufferSet();
r_tStaticTestDone(CLK			:= (iCompareStaticSM = 110));
r_tSetDUTVal();
tonReadWait(PT		:= tTestTime);
tonConvert(PT		:= tTestTime);
tonWriteCopyWait(PT	:= tWriteWaitTime);
tonTestIterGap(PT	:= tTestTime);
tTestTime			:= T#80MS;
//just an example one
tWriteWaitTime		:= T#10MS; // same as the tOffDelay set to the input debounce FB
//DMX DUT Channels, Software 0-255 
//DMX Config Channels, Software, 256-511
//DMX DUT Channels, Hardware 1-256
//DMX Config Channels, Hardware, 257-512

//Interface Link - continued - DMXTest Local Vars

//"Config Complete" Expctd Buffer, and "Config Complete" Received Buffer; then Global Comparison is like 'masking' all but one channel at a time;

CASE iParseFile OF

0:
IF P_TextModeRead.r_tFileChg.Q THEN
	xFileImported		:= FALSE;	
	iParseFile			:= 5;
END_IF

5:
IF P_TextModeRead.fbFileGets.bEOF THEN
	uiForLoopRecipe	:= 0; // Reset the iterator used in the next state of the SM
	iParseFile		:= 10;
END_IF
	
10://At first check for any recipe items specified in the file;
//Load the recipe data into respective arrays
//For recipe indices = 0 to 255, parse the file to read the recipe index, DMX channel, and channel type
FOR uiForLoopRecipe := 0 TO gc.uiDUTConfigCountSplit BY 1 DO
	//Read the Recipe Index
	arr_uiRecipeIndexTmp[uiForLoopRecipe]		:= STRING_TO_UINT(P_TextModeRead.database[uiForLoopRecipe,0]);
	//Read the DMX Channel for the DUT
	arruiDMXChDUTTmp[uiForLoopRecipe]			:= STRING_TO_UINT(P_TextModeRead.database[uiForLoopRecipe,1]);
	//Read the type of Channel on the DUT
	arrsDUTChTypeTmp[uiForLoopRecipe]			:= P_TextModeRead.database[uiForLoopRecipe,2];
END_FOR
//Stash the values from temp (inside FOR loop) to other arrays
arr_uiRecipeIndex	:= arr_uiRecipeIndexTmp;
arruiDMXChDUT		:= arruiDMXChDUTTmp;
arrsDUTChType		:= arrsDUTChTypeTmp;

//If the 'TextModeRead' re-enters 'Ready' state then advance this SM
IF P_TextModeRead.step = 0 THEN
	xFileImported		:= TRUE;
	iParseFile			:= 0;	
END_IF

END_CASE

CASE iSetConfig OF

//Don't look at the P_TextRead; evaluate on the arrays you just imported

0:
IF r_tSetConfig.Q THEN
	iSetConfig			:= 10;	
END_IF

10://Read the string that is loaded from file reader; pass value to DMX Function Block, at the appropriate Config index
//This is the setting to control the position of the 'config' relays on the tester
//Ensure that the declared arrays are sufficiently long to handle the max conceivable value (512 x 2, in this case?)
FOR uiForLoopRecipe := 0 TO gc.uiDUTConfigCountSplit BY 1 DO
	IF (arruiDMXChDUT[uiForLoopRecipe] <> 0) THEN
		//Set the config routing := NPN
		arr_usiRecipeSettingTmp[(uiForLoopRecipe+gc.uiChannelSplitCount)]	:= 255;
	ELSIF (arruiDMXChDUT[uiForLoopRecipe] = 0) THEN
		//Set the config routing := PNP
		arr_usiRecipeSettingTmp[(uiForLoopRecipe+gc.uiChannelSplitCount)]	:= 0;
	END_IF	
END_FOR
//Stash the values from temp (inside FOR loop) to other arrays
arr_usiRecipeSetting	:= arr_usiRecipeSettingTmp;

	iSetConfig			:= 20;	

20://Iterate over the config listings to create indices for what must be tested static (power, ground), and what must be tested sequentially (channels)
uiLoopIterDMXDUTArraySeq	:= 0;
uiLoopIterTestArrSeq		:= 0;
//Zero out the array that is copied to in the next state of the SM
FOR uiForLoopZeroStorageArray	:= 0 TO gc.uiMaxNrOfDMXChannel BY 1 DO
	arruiSeqTestIndicesTmp[uiForLoopZeroStorageArray]	:= 0;
END_FOR
//Stash the values from temp (inside FOR loop) to other arrays
arruiSeqTestIndices		:= arruiSeqTestIndicesTmp;
iSetConfig				:= 40;	

40:
//For any 'DMX'-type channels with an assigned channel # (from the recipe), then copy only those elements to another array
//These are elements that are tested sequentially - once - so this includes Dry Contacts but not Motors
REPEAT
	IF ((arrsDUTChType[uiLoopIterDMXDUTArraySeq] = 'DMX') OR (arrsDUTChType[uiLoopIterDMXDUTArraySeq] = '24V')) AND (arruiDMXChDUT[uiLoopIterDMXDUTArraySeq] <> 0) THEN
		MEMCPY(srcAddr:=ADR(arruiDMXChDUT[uiLoopIterDMXDUTArraySeq]),destAddr:=ADR(arruiSeqTestIndicesTmp[uiLoopIterDMXDUTArraySeq]),n:=SIZEOF(arruiDMXChDUT[uiLoopIterDMXDUTArraySeq])); //UINT = 4 bytes?
//		uiLoopIterTestArrSeq		:= uiLoopIterTestArrSeq+1;
	END_IF
	uiLoopIterDMXDUTArraySeq	:= uiLoopIterDMXDUTArraySeq+1;
UNTIL 
(uiLoopIterDMXDUTArraySeq = gc.uiMaxNrOfDMXChannel)
END_REPEAT
//Stash the values from temp (inside FOR loop) to other arrays
arruiSeqTestIndices		:= arruiSeqTestIndicesTmp;

iSetConfig					:= 50;	

50:
//Use different iterators - set them to 0 prior to use
uiLoopIterDMXDUTArrayM		:= 0;
uiLoopIterTestArrM			:= 0;
//Zero out the array that is copied to in the next state of the SM
FOR uiForLoopZeroStorageArray	:= 0 TO gc.uiMaxNrOfDMXChannel BY 1 DO
	arruiMotorTestIndicesTmp[uiForLoopZeroStorageArray]	:= 0;
END_FOR
//Stash the values from temp (inside FOR loop) to other arrays
arruiMotorTestIndices	:= arruiMotorTestIndicesTmp;

iSetConfig					:= 60;	

60:
//Motors - Type code "M" - must be tested both in the PNP & NPN inputs
//This array easily provides the indexing for which channels the motors are on
REPEAT
	IF (arrsDUTChType[uiLoopIterDMXDUTArrayM] = 'M') AND (arruiDMXChDUT[uiLoopIterDMXDUTArrayM] <> 0)  THEN
		MEMCPY(srcAddr:=ADR(arruiDMXChDUT[uiLoopIterDMXDUTArrayM]),destAddr:=ADR(arruiMotorTestIndicesTmp[uiLoopIterDMXDUTArrayM]),n:=SIZEOF(arruiDMXChDUT[uiLoopIterDMXDUTArrayM])); //UINT = 4 bytes?
//		uiLoopIterTestArrM		:= uiLoopIterTestArrM+1;
	END_IF
	uiLoopIterDMXDUTArrayM	:= uiLoopIterDMXDUTArrayM+1;
UNTIL 
(uiLoopIterDMXDUTArrayM = gc.uiMaxNrOfDMXChannel)
END_REPEAT
//Stash the values from temp (inside FOR loop) to other arrays
arruiMotorTestIndices	:= arruiMotorTestIndicesTmp;

iSetConfig		:= 70;

70:
//Use different iterators - set them to 0 prior to use
uiLoopIterDUTArray24V		:= 0;
uiLoopIterTestArr24V		:= 0;
//Zero out the array that is copied to in the next state of the SM
FOR uiForLoopZeroStorageArray	:= 0 TO gc.uiMaxNrOfDMXChannel BY 1 DO
	arrui24VTestIndicesTmp[uiForLoopZeroStorageArray]	:= 0;
END_FOR
//Stash the values from temp (inside FOR loop) to other arrays
arrui24VTestIndices		:= arrui24VTestIndicesTmp;

iSetConfig				:= 80;

80:
//24V - Type code "24V" - is tested per static config
//This array easily provides the indexing for which channels the 24V are on
REPEAT
	IF (arrsDUTChType[uiLoopIterDUTArray24V] = '24V') AND (arruiDMXChDUT[uiLoopIterDUTArray24V] = 0) THEN
		MEMCPY(srcAddr:=ADR(arr_uiRecipeIndex[uiLoopIterDUTArray24V]),destAddr:=ADR(arrui24VTestIndicesTmp[uiLoopIterDUTArray24V]),n:=SIZEOF(arr_uiRecipeIndex[uiLoopIterDUTArray24V])); //UINT = 2 bytes?
//		uiLoopIterTestArr24V	:= uiLoopIterTestArr24V +1;
	END_IF
	uiLoopIterDUTArray24V	:= uiLoopIterDUTArray24V+1;
UNTIL 
(uiLoopIterDUTArray24V = gc.uiDUTConfigCountSplit)
END_REPEAT
//Stash the values from temp (inside FOR loop) to other arrays
arrui24VTestIndices	:= arrui24VTestIndicesTmp;

iSetConfig		:= 90;

90://Clear Iterators for GND channel indexing
//Use different iterators - set them to 0 prior to use
uiLoopIterDUTArrayGND		:= 0;
uiLoopIterTestArrGND		:= 0;
//Zero out the array that is copied to in the next state of the SM
FOR uiForLoopZeroStorageArray	:= 0 TO gc.uiMaxNrOfDMXChannel BY 1 DO
	arruiGNDTestIndicesTmp[uiForLoopZeroStorageArray]	:= 0;
END_FOR
//Stash the values from temp (inside FOR loop) to other arrays
arruiGNDTestIndices		:= arruiGNDTestIndicesTmp;

iSetConfig				:= 100;

100:
//Ground - Type code "GND" - is tested per static config
//This array easily provides the indexing for which channels the 24V are on
REPEAT
	IF (arrsDUTChType[uiLoopIterDUTArrayGND] = 'GND') AND (arruiDMXChDUT[uiLoopIterDUTArrayGND] = 0) THEN
		MEMCPY(srcAddr:=ADR(arr_uiRecipeIndex[uiLoopIterDUTArrayGND]),destAddr:=ADR(arruiGNDTestIndicesTmp[uiLoopIterDUTArrayGND]),n:=SIZEOF(arr_uiRecipeIndex[uiLoopIterDUTArrayGND])); //UINT = 4 bytes?
//		uiLoopIterTestArrGND	:= uiLoopIterTestArrGND+1;
	END_IF
	uiLoopIterDUTArrayGND	:= uiLoopIterDUTArrayGND+1;
UNTIL 
(uiLoopIterDUTArrayGND = gc.uiDUTConfigCountSplit)
END_REPEAT
//Stash the values from temp (inside FOR loop) to other arrays
arruiGNDTestIndices	:= arruiGNDTestIndicesTmp;

iSetConfig				:= 110;

//Copy of state30
110://Iterate over the config listings to create indices for what must be tested static (power, ground), and what must be tested sequentially (channels)
uiLoopIterDMXDUTArraySeq		:= 0;
uiLoopIterTestArrSeq			:= 0;
//Zero out the array that is copied to in the next state of the SM
FOR uiForLoopZeroStorageArray	:= 0 TO gc.uiMaxNrOfDMXChannel BY 1 DO
	arruiSeqTestIndicesDMXTmp[uiForLoopZeroStorageArray]	:= 0;
	arruiSeqTestIndicesDMXSW[uiForLoopZeroStorageArray]		:= 0;
END_FOR
//Stash the values from temp (inside FOR loop) to other arrays
arruiSeqTestIndicesDMX			:= arruiSeqTestIndicesDMXTmp;
iSetConfig						:= 120;	

120://Effectively a copy of state40
//For any 'DMX'-type channels with an assigned channel # (from the recipe), then copy only those elements to another array
//These are elements that are tested sequentially - once - so this includes Dry Contacts but not Motors
REPEAT
	IF (arrsDUTChType[uiLoopIterDMXDUTArraySeq] = 'DMX') AND (arruiDMXChDUT[uiLoopIterDMXDUTArraySeq] <> 0) THEN
		MEMCPY(srcAddr:=ADR(arruiDMXChDUT[uiLoopIterDMXDUTArraySeq]),destAddr:=ADR(arruiSeqTestIndicesDMXTmp[uiLoopIterDMXDUTArraySeq]),n:=SIZEOF(arr_uiRecipeIndex[uiLoopIterDUTArrayGND])); //UINT = 4 bytes?
//		uiLoopIterTestArrSeq		:= uiLoopIterTestArrSeq+1;
	END_IF
	uiLoopIterDMXDUTArraySeq		:= uiLoopIterDMXDUTArraySeq+1;
UNTIL 
(uiLoopIterDMXDUTArraySeq = gc.uiMaxNrOfDMXChannel)
END_REPEAT
//Stash the values from temp (inside FOR loop) to other arrays
arruiSeqTestIndicesDMX				:= arruiSeqTestIndicesDMXTmp;

//Set the recipe addresses one lower for 'SW'-Software-because software indexes from 0, not 1
FOR uiCounter8	:= 0 TO gc.uiMaxNrDMXTestCh BY 1 DO
	IF arruiSeqTestIndicesDMX[uiCounter8] <> 0 THEN
		arruiSeqTestIndicesDMXSW[uiCounter8]	:= arruiSeqTestIndicesDMX[uiCounter8] - 1;	
	END_IF
END_FOR

iSetConfig							:= 130;	

//Copy of state30
130://Iterate over the config listings to create indices for what must be tested static (power, ground), and what must be tested sequentially (channels)
uiLoopIterDMXDUTArraySeq		:= 0;
uiLoopIterTestArrSeq			:= 0;
//Zero out the array that is copied to in the next state of the SM
FOR uiForLoopZeroStorageArray	:= 0 TO gc.uiMaxNrOfDMXChannel BY 1 DO
	arruiSeqTestIndicesDCTmp[uiForLoopZeroStorageArray]	:= 0;
END_FOR
//Stash the values from temp (inside FOR loop) to other arrays
arruiSeqTestIndicesDC			:= arruiSeqTestIndicesDCTmp;
iSetConfig						:= 140;	

140:
//For any 'DMX'-type channels with an assigned channel # (from the recipe), then copy only those elements to another array
//These are elements that are tested sequentially - once - so this includes Dry Contacts but not Motors
REPEAT
	IF (arrsDUTChType[uiLoopIterDMXDUTArraySeq] = '24V') AND (arruiDMXChDUT[uiLoopIterDMXDUTArraySeq] <> 0) THEN
		MEMCPY(srcAddr:=ADR(arruiDMXChDUT[uiLoopIterDMXDUTArraySeq]),destAddr:=ADR(arruiSeqTestIndicesDCTmp[uiLoopIterDMXDUTArraySeq]),n:=SIZEOF(arruiDMXChDUT[uiLoopIterDMXDUTArraySeq])); //UINT = 4 bytes?
//		uiLoopIterTestArrSeq		:= uiLoopIterTestArrSeq+1;
	END_IF
	uiLoopIterDMXDUTArraySeq		:= uiLoopIterDMXDUTArraySeq+1;
UNTIL 
(uiLoopIterDMXDUTArraySeq = gc.uiMaxNrOfDMXChannel)
END_REPEAT
//Stash the values from temp (inside FOR loop) to other arrays
arruiSeqTestIndicesDC				:= arruiSeqTestIndicesDCTmp;

iSetConfig							:= 0;	

END_CASE


//Set the config of the 'routing' channels
IF r_tSetConfig.Q THEN
	g_ast.DMXHWOut	:= g_ast.DMXPhysOut;
//	xConfigSet		:= TRUE;
END_IF


// For manual setting of channels from the Visualization - NOTE! This stamps over any other values set for the lower 256 channels (DUT)
CASE iSetDUTSM OF
	
0:
IF r_tSetDUTVal.Q THEN
	iSetDUTSM		:= 10;
END_IF

10:
FOR uiForLoopDUTIter := 0 TO gc.uiDUTConfigCountSplit BY 1 DO
	g_ast.DMXHWOut[uiForLoopDUTIter] 	:= usiDUTVal;
END_FOR
//g_ast.DMXHWOut					:= g_ast.DMXPhysOut;

IF NOT r_tSetDUTVal.Q THEN
	iSetDUTSM	:= 0;
END_IF

END_CASE


CASE iSetExpctdBufferSM OF
	
0://If there is a trigger to set the test config, create a new 'Expctd' buffer
IF r_tSetExpectedBuff.Q THEN
	r_tExpectedBufferSet.CLK	:= FALSE;
	//Clear the existing buffers
	FOR uiForLoopClearExpctd := 0 TO gc.uiMaxNrOfDMXChannel BY 1 DO
		arrxExpctdPNP[uiForLoopClearExpctd]	:= 0;
		arrxExpctdNPN[uiForLoopClearExpctd]	:= 0;
	END_FOR
	iSetExpctdBufferSM			:= 10;
END_IF

10: // Set Expected Buffers per Recipe Files
FOR uiLoopExpctdIndex := 0 TO gc.uiMaxNrOfDMXChannel BY 1 DO
	IF (arr_usiRecipeSetting[uiLoopExpctdIndex] <= 127) THEN
		arrxExpctdPNP[arr_uiRecipeIndex[uiLoopExpctdIndex]]		:= TRUE; 
		arrxExpctdNPN[arr_uiRecipeIndex[uiLoopExpctdIndex]]		:= FALSE;
	ELSIF (arr_usiRecipeSetting[uiLoopExpctdIndex] > 127) THEN
		arrxExpctdPNP[arr_uiRecipeIndex[uiLoopExpctdIndex]]		:= FALSE;
		arrxExpctdNPN[arr_uiRecipeIndex[uiLoopExpctdIndex]]		:= TRUE; 
	END_IF
	//Zero out Expected, type-specific index buffers
	arrxExpctdTmpPNP24V[uiLoopExpctdIndex] 					:= 0;
	arrxExpctdTmpNPN24V[uiLoopExpctdIndex] 					:= 0;
	arrxExpctdTmpPNPGND[uiLoopExpctdIndex] 					:= 0;
	arrxExpctdTmpNPNGND[uiLoopExpctdIndex] 					:= 0;
END_FOR

r_tExpectedBufferSet.CLK	:= TRUE;
iSetExpctdBufferSM			:= 0;

END_CASE

CASE iReindexExpctedBufferSM OF
	
0:
IF r_tExpectedBufferSet.Q THEN
	iReindexExpctedBufferSM	:= 10;
END_IF

10://Copy the contents of Expected Buffer to a different Buffer, starting at array address 0 - only the channels that have a hardware input index
MEMCPY(srcAddr:=ADR(arrxExpctdPNP[gc.uiChannelSplitCount]),destAddr:=ADR(arrxExpctdTmpPNP[cuiMinDUTIndex]),n:=gc.uiChannelsUT);
MEMCPY(srcAddr:=ADR(arrxExpctdNPN[gc.uiChannelSplitCount]),destAddr:=ADR(arrxExpctdTmpNPN[cuiMinDUTIndex]),n:=gc.uiChannelsUT);

iReindexExpctedBufferSM	:= 20;

20:
//And create the comparison Expected Buffer for Static Test - 24V & GND indices
FOR uiCounter5 := 0 TO gc.uiMaxNrDMXTestCh BY 1 DO
	IF arrui24VTestIndices[uiCounter5] <> 0 THEN	
		MEMCPY(srcAddr:=ADR(arrxExpctdTmpPNP[arrui24VTestIndices[uiCounter5]]),destAddr:=ADR(arrxExpctdTmpPNP24V[arrui24VTestIndices[uiCounter5]]),n:=SIZEOF(arrxExpctdTmpPNP[arrui24VTestIndices[uiCounter5]])); //bytes
		MEMCPY(srcAddr:=ADR(arrxExpctdTmpNPN[arrui24VTestIndices[uiCounter5]]),destAddr:=ADR(arrxExpctdTmpNPN24V[arrui24VTestIndices[uiCounter5]]),n:=SIZEOF(arrxExpctdTmpNPN[arrui24VTestIndices[uiCounter5]])); //bytes
	END_IF
	
	IF arruiGNDTestIndices[uiCounter5] <> 0 THEN	
		MEMCPY(srcAddr:=ADR(arrxExpctdTmpPNP[arruiGNDTestIndices[uiCounter5]]),destAddr:=ADR(arrxExpctdTmpPNPGND[arruiGNDTestIndices[uiCounter5]]),n:=SIZEOF(arrxExpctdTmpPNP[arruiGNDTestIndices[uiCounter5]])); //bytes
		MEMCPY(srcAddr:=ADR(arrxExpctdTmpNPN[arruiGNDTestIndices[uiCounter5]]),destAddr:=ADR(arrxExpctdTmpNPNGND[arruiGNDTestIndices[uiCounter5]]),n:=SIZEOF(arrxExpctdTmpNPN[arruiGNDTestIndices[uiCounter5]])); //bytes
	END_IF	
END_FOR

iReindexExpctedBufferSM	:= 0;

END_CASE


CASE iCompareStaticSM OF
	
0: // If test is triggered by user
IF rt_RunStaticTest.Q THEN
	xStatTestInProgress						:= TRUE;
	uiLoopRcvIndex							:= cuiMinDUTIndex; 
	iCompareStaticSM						:= 10;
END_IF

10: // Zero out all comparison buffers before each comparison
//IF (uiLoopRcvIndex=0) THEN
	IF xStatTestInProgress THEN
		//by default, Counter = 0 at the first initialization; it is reset at the end of this State Machine
		//Clear Storage Buffers pre-test to ensure no old data interferes with current test
		FOR uiCounter4 := 0 TO gc.uiDUTConfigCountSplit BY 1 DO
			arrxRcvdBufferPNP24V[uiCounter4]	:= 0;		
			arrxRcvdBufferNPN24V[uiCounter4]	:= 0;		
			arrxRcvdBufferPNPGND[uiCounter4]	:= 0;		
			arrxRcvdBufferNPNGND[uiCounter4]	:= 0;		
			g_ast.DMX[uiCounter4].IQ.xCmdOff	:= TRUE;	
		END_FOR
	iCompareStaticSM				:= 20;
	END_IF
(*
ELSIF (uiLoopRcvIndex>0) THEN
	IF xStatTestInProgress AND tonTestIterGap.Q THEN
		tonTestIterGap.IN	:= FALSE;
		//by default, Counter = 0 at the first initialization; it is reset at the end of this State Machine
		//Clear Storage Buffers pre-test to ensure no old data interferes with current test
		FOR uiCounter4 := 0 TO gc.uiDUTConfigCountSplit BY 1 DO
			arrxRcvdBufferPNP24V[uiCounter4]	:= 0;		
			arrxRcvdBufferNPN24V[uiCounter4]	:= 0;		
			arrxRcvdBufferPNPGND[uiCounter4]	:= 0;		
			arrxRcvdBufferNPNGND[uiCounter4]	:= 0;		
		END_FOR
	iCompareStaticSM				:= 30; // don't write the hardware value (skip 20)
	END_IF
END_IF
*)
	
20:	
//write 'hardware-clear' state 
g_ast.DMXHWOut					:= g_ast.DMXPhysOut;
iCompareStaticSM				:= 30;

30: //Set the Expected Mask & write data to controller
(*
IF uiLoopRcvIndex <> 0 THEN
//	g_ast.DMX[uiLoopRcvIndex].IQ.xCmdOn			:= TRUE;
	FOR uiCounter3 := cuiMinDUTIndex TO gc.uiMaxNrDMXTestCh BY 1 DO
		IF uiCounter3 <> uiLoopRcvIndex THEN
			g_ast.DMX[uiCounter3].IQ.xCmdOff	:= TRUE;	
		END_IF
	END_FOR
	iCompareStaticSM		:= 40;
ELSE //uiLoopRcvIndex = 0
	*)
tonWriteCopyWait.IN		:= TRUE;
iCompareStaticSM		:= 50;
//END_IF

40:
//Write DMX channels
(*
g_ast.DMXHWOut			:= g_ast.DMXPhysOut;
tonWriteCopyWait.IN		:= TRUE;
iCompareStaticSM		:= 50;
*)

50:
IF tonWriteCopyWait.Q THEN
	tonWriteCopyWait.IN	:= FALSE;
	iCompareStaticSM	:= 60;
END_IF

60:
FOR uiCounter4 := 0 TO gc.uiMaxNrDMXTestCh BY 1 DO

//IF there is an index for a '24V' element, then copy that element's value to a new pair of arrays, for 'Received'

	IF arrui24VTestIndices[uiCounter4] <> 0 THEN

		arrudiStaticCopyResultPNP24V[arrui24VTestIndices[uiCounter4]]	:= MEMCPY(srcAddr:=ADR(g_ast.arrInputPNP[arrui24VTestIndices[uiCounter4]]),destAddr:=ADR(arrxRcvdBufferPNP24V[arrui24VTestIndices[uiCounter4]]),n:=SIZEOF(g_ast.arrInputPNP[arrui24VTestIndices[uiCounter4]])); //bytes
		arrudiStaticCopyResultNPN24V[arrui24VTestIndices[uiCounter4]]	:= MEMCPY(srcAddr:=ADR(g_ast.arrInputNPN[arrui24VTestIndices[uiCounter4]]),destAddr:=ADR(arrxRcvdBufferNPN24V[arrui24VTestIndices[uiCounter4]]),n:=SIZEOF(g_ast.arrInputNPN[arrui24VTestIndices[uiCounter4]])); //bytes)

	END_IF

//IF there is an index for a 'GND' element, then copy that element's value to a new pair of arrays, for 'Received'

	IF arruiGNDTestIndices[uiCounter4] <> 0 THEN

		arrudiStaticCopyResultPNPGND[arruiGNDTestIndices[uiCounter4]]	:= MEMCPY(srcAddr:=ADR(g_ast.arrInputPNP[arruiGNDTestIndices[uiCounter4]]),destAddr:=ADR(arrxRcvdBufferPNPGND[arruiGNDTestIndices[uiCounter4]]),n:=SIZEOF(g_ast.arrInputPNP[arruiGNDTestIndices[uiCounter4]])); //bytes
		arrudiStaticCopyResultNPNGND[arruiGNDTestIndices[uiCounter4]]	:= MEMCPY(srcAddr:=ADR(g_ast.arrInputNPN[arruiGNDTestIndices[uiCounter4]]),destAddr:=ADR(arrxRcvdBufferNPNGND[arruiGNDTestIndices[uiCounter4]]),n:=SIZEOF(g_ast.arrInputNPN[arruiGNDTestIndices[uiCounter4]])); //bytes)
	
	END_IF
	
END_FOR

iCompareStaticSM			:= 70;

70:
tonReadWait.IN				:= TRUE;
iCompareStaticSM			:= 80;

80: // if wait completed, set the bit for conversion high
//Conversion Function call
IF tonReadWait.Q THEN
	tonReadWait.IN					:= FALSE;
	iCompareStaticSM				:= 90;
END_IF

90:
//Run Comparos
//Individual Channels comparison
FOR uiCounter6	:= 0 TO gc.uiMaxNrDMXTestCh BY 1 DO 
	arr_diTestStaticPNP24V[uiCounter6]		:= MEMCMP(pBuf1:=ADR(arrxExpctdTmpPNP24V[uiCounter6]),pBuf2:=ADR(arrxRcvdBufferPNP24V[uiCounter6]),n:=SIZEOF(arrxExpctdTmpPNP24V[uiCounter6]));
	arr_diTestStaticNPN24V[uiCounter6]		:= MEMCMP(pBuf1:=ADR(arrxExpctdTmpNPN24V[uiCounter6]),pBuf2:=ADR(arrxRcvdBufferNPN24V[uiCounter6]),n:=SIZEOF(arrxExpctdTmpNPN24V[uiCounter6]));
	arr_diTestStaticPNPGND[uiCounter6]		:= MEMCMP(pBuf1:=ADR(arrxExpctdTmpPNPGND[uiCounter6]),pBuf2:=ADR(arrxRcvdBufferPNPGND[uiCounter6]),n:=SIZEOF(arrxExpctdTmpPNPGND[uiCounter6]));
	arr_diTestStaticNPNGND[uiCounter6]		:= MEMCMP(pBuf1:=ADR(arrxExpctdTmpNPNGND[uiCounter6]),pBuf2:=ADR(arrxRcvdBufferNPNGND[uiCounter6]),n:=SIZEOF(arrxExpctdTmpNPNGND[uiCounter6]));
END_FOR

//Complete Buffer
diTestStaticPNP24V		:= MEMCMP(pBuf1:=ADR(arrxExpctdTmpPNP24V[cuiMinDUTIndex]),pBuf2:=ADR(arrxRcvdBufferPNP24V[cuiMinDUTIndex]),n:=gc.uiChannelsUT);
diTestStaticNPN24V		:= MEMCMP(pBuf1:=ADR(arrxExpctdTmpNPN24V[cuiMinDUTIndex]),pBuf2:=ADR(arrxRcvdBufferNPN24V[cuiMinDUTIndex]),n:=gc.uiChannelsUT);
diTestStaticPNPGND		:= MEMCMP(pBuf1:=ADR(arrxExpctdTmpPNPGND[cuiMinDUTIndex]),pBuf2:=ADR(arrxRcvdBufferPNPGND[cuiMinDUTIndex]),n:=gc.uiChannelsUT);
diTestStaticNPNGND		:= MEMCMP(pBuf1:=ADR(arrxExpctdTmpNPNGND[cuiMinDUTIndex]),pBuf2:=ADR(arrxRcvdBufferNPNGND[cuiMinDUTIndex]),n:=gc.uiChannelsUT);

iCompareStaticSM				:= 105;

(*
100: // If counter is equal to the max # of test channels, reset it; turn off the DMX channels that were turned on in the course of the test
IF (uiLoopRcvIndex = gc.uiMaxNrDMXTestCh) THEN
	rt_RunStaticTest.CLK			:= TRUE;
	iCompareStaticSM				:= 110;
ELSE
	uiLoopRcvIndex				:= uiLoopRcvIndex +1;
	//Next iteration
	tonTestIterGap.IN			:= TRUE;
	iCompareStaticSM			:= 10;
 (*iCounter <> gc.usiMaxNrOfChannels*)
END_IF
*)

105:
//Retrieving the discrepant indices for display on HMI
FOR uiVisuIndex := 0 TO gc.uiMaxNrDMXTestCh BY 1 DO
	IF (arr_diTestStaticPNP24V[uiVisuIndex] <> 0) THEN
		arrVisu_diTestResult[uiVisuIndex]	:= uiVisuIndex;	
	ELSIF (arr_diTestStaticNPNGND[uiVisuIndex] <> 0) THEN
		arrVisu_diTestResult[uiVisuIndex]	:= uiVisuIndex;	
	END_IF
END_FOR

iCompareStaticSM				:= 110;
	
110:
xStatTestInProgress				:= FALSE;
iCompareStaticSM				:= 120;

120:
IF rt_ResetTest.Q AND NOT rt_RunStaticTest.Q THEN
	FOR uiCounter2 := 0 TO gc.uiMaxNrDMXTestCh BY 1 DO 
		arr_diTestStaticPNP24V[uiCounter2]		:= 0;
		arr_diTestStaticNPN24V[uiCounter2]		:= 0;
		arr_diTestStaticPNPGND[uiCounter2]		:= 0;
		arr_diTestStaticNPNGND[uiCounter2]		:= 0;
	END_FOR
	diCompTestResult							:= 0;
	iCompareStaticSM							:= 0; (* reset to beginning *)
END_IF

END_CASE


//Linked to the Visualization Table
//FOR uiVisuIndex := 0 TO gc.uiMaxNrDMXTestCh BY 1 DO
	//	arrVisu_diTestResult[0,uiVisuIndex]	:= g_ast.DMXHWOut[uiVisuIndex]; //Sent
	//	arrVisu_diTestResult[1,uiVisuIndex]	:= arrbySclPNP[uiVisuIndex]; //Received
	//	arrVisu_diTestResult[2,uiVisuIndex]	:= arr_diTestResultPNP[uiVisuIndex]; //Result of Comparison
	//	arrVisu_diTestResult[3,uiVisuIndex]	:= arr_diTestResultNPN[uiVisuIndex]; //Result of Comparison
//END_FOR



//IF diCompTestResultTemp = -1 OR diCompTestResultTemp = 1 THEN
//	diCompTestResult	:= diCompTestResultTemp;
//END_IF

ACTION InvertRecipeSettings:
R_TInvertRecipe();

CASE iInvertRecipeSM OF
	
0:
IF R_TInvertRecipe.Q THEN
	iInvertRecipeSM		:= 10;
END_IF

10:
FOR uiRecipeInvertIter := uiStartingIndex TO uiEndingIndex BY 1 DO 
	IF arr_usiRecipeSetting[uiRecipeInvertIter] = 0 THEN
		arr_usiRecipeSetting[uiRecipeInvertIter]	:= 255;
	ELSIF arr_usiRecipeSetting[uiRecipeInvertIter] <> 0 THEN
		arr_usiRecipeSetting[uiRecipeInvertIter]	:= 0;
	END_IF
END_FOR

iInvertRecipeSM		:= 20;

20:
IF NOT R_TInvertRecipe.Q THEN
	iInvertRecipeSM		:= 0;
END_IF

END_CASE
END_ACTION

ACTION SeqTestMotor:

END_ACTION

ACTION SeqTestOnce:
//Run Once - DMX Channels only for now

rt_RunSeqTestOnce();
rt_ResetTestSeq();

CASE iCompareSeq[ENUM_SeqSM.Once] OF
	
0: // If test is triggered by user
//Trigger should be something like 
IF rt_RunSeqTestOnce.Q THEN
	xDMXSeqTestInProgressOnce				:= TRUE;
	uiLoopRcvIndex							:= cuiMinDUTIndex; 
	iCompareSeq[ENUM_SeqSM.Once]			:= 10;
END_IF

10: // Zero out all comparison buffers before each comparison
IF (uiLoopRcvIndex=0) THEN
	IF xDMXSeqTestInProgressOnce THEN
//by default, Counter = 0 at the first initialization; it is reset at the end of this State Machine
//Clear Storage Buffers pre-test to ensure no old data interferes with current test
		FOR uiCounter4 := 0 TO gc.uiMaxNrDMXTestCh BY 1 DO
			arrxExpctdTmpPNPSeqDMX[uiCounter4]		:= 0;		//should be all 0s ; PNP<>DMX
			arrxExpctdTmpNPNSeqDMX[uiCounter4]		:= 0;
//			arrxExpctdTmpPNPSeqDC[uiCounter4]		:= 0;		
//			arrxExpctdTmpNPNSeqDC[uiCounter4]		:= 0;
			arrxRcvdBufferPNPSeq[uiCounter4]		:= 0;		//should be all 0s too ; PNP<>DMX	
			arrxRcvdBufferNPNSeq[uiCounter4]		:= 0;			
			g_ast.DMX[uiCounter4].IQ.xCmdOff		:= TRUE;	
		END_FOR
	iCompareSeq[ENUM_SeqSM.Once]					:= 20;
	END_IF
ELSIF (uiLoopRcvIndex>0) THEN // to avoid 
	IF xDMXSeqTestInProgressOnce AND tonTestIterGap.Q THEN
		tonTestIterGap.IN	:= FALSE;
		//by default, Counter = 0 at the first initialization; it is reset at the end of this State Machine
		//Clear Storage Buffers pre-test to ensure no old data interferes with current test
		FOR uiCounter4 := 0 TO gc.uiMaxNrDMXTestCh BY 1 DO
			arrxExpctdTmpPNPSeqDMX[uiCounter4]		:= 0;		//should be all 0s - PNP<>DMX
			arrxExpctdTmpNPNSeqDMX[uiCounter4]		:= 0;
			arrxRcvdBufferPNPSeq[uiCounter4]		:= 0;		
			arrxRcvdBufferNPNSeq[uiCounter4]		:= 0;
		END_FOR
		
	iCompareSeq[ENUM_SeqSM.Once]					:= 20; // don't write the hardware value (skip 20)
	END_IF	
END_IF
	
20:	
//write 'hardware-clear' state 
g_ast.DMXHWOut									:= g_ast.DMXPhysOut;

iCompareSeq[ENUM_SeqSM.Once]					:= 25;

25:
//Copy static test indices from Expected_Static - as these should still be used for comparisons
//	IF (arrui24VTestIndices[uiCounter4] <> 0) THEN	
//		MEMCPY(srcAddr:=ADR(arrxExpctdTmpPNP24V[cuiMinDUTIndex]),destAddr:=ADR(arrxExpctdTmpPNPSeqDMX[cuiMinDUTIndex]),n:=gc.uiChannelsUT);
FOR uiCounter4 := 0 TO gc.uiMaxNrDMXTestCh BY 1 DO
	arrxExpctdTmpPNPSeqDMX[uiCounter4]		:= arrxExpctdTmpPNP24V[uiCounter4];
	arrxExpctdTmpNPNSeqDMX[uiCounter4]		:= arrxExpctdTmpNPNGND[uiCounter4];
END_FOR

iCompareSeq[ENUM_SeqSM.Once]					:= 30;

30: //Set the Expected Mask & write data to controller
//Write the first index from the specified array of indices
//MEMCPY(srcAddr:=ADR(arrxExpctdTmpNPN[arruiSeqTestIndicesDMX[uiLoopRcvIndex]]),destAddr:=ADR(arrxExpctdTmpNPNSeqDMX[arruiSeqTestIndicesDMX[uiLoopRcvIndex]]),n:=SIZEOF(arrxExpctdTmpNPN[arruiSeqTestIndicesDMX[uiLoopRcvIndex]]));	

//This line copies only the value of the current iterator's index in the DMX Channel Array
arrxExpctdTmpNPNSeqDMX[uiLoopRcvIndex]	:= arrxExpctdTmpNPN[uiLoopRcvIndex];

iCompareSeq[ENUM_SeqSM.Once]			:= 35;

35:
IF (arruiSeqTestIndicesDMXSW[uiLoopRcvIndex] <> 0) THEN
//Also copy this specific channel index value to the comparison array
	
//Don't copy PNP indices for DMX; this doesn't generally make sense
//	MEMCPY(srcAddr:=ADR(arrxExpctdTmpPNP[arruiSeqTestIndicesDMX[uiLoopRcvIndex]]),destAddr:=ADR(arrxExpctdTmpPNPSeqDMX[arruiSeqTestIndicesDMX[uiLoopRcvIndex]]),n:=1);
	
	//CmdOn - command on - that respective channel
	g_ast.DMX[arruiSeqTestIndicesDMXSW[uiLoopRcvIndex]].IQ.xCmdOn			:= TRUE;
	//and turn off all others
	FOR uiCounter3 := cuiMinDUTIndex TO gc.uiMaxNrDMXTestCh BY 1 DO
		IF uiCounter3 <> arruiSeqTestIndicesDMXSW[uiLoopRcvIndex] THEN
			g_ast.DMX[uiCounter3].IQ.xCmdOff	:= TRUE;	
		END_IF
	END_FOR
END_IF

iCompareSeq[ENUM_SeqSM.Once]		:= 40;

40:
//Write to hardware
g_ast.DMXHWOut							:= g_ast.DMXPhysOut;
//tonWriteCopyWait.IN						:= TRUE;
iCompareSeq[ENUM_SeqSM.Once]			:=	60;

(*
50:

//Timer marks end of sampling period; reset timer
IF tonWriteCopyWait.Q THEN
	tonWriteCopyWait.IN					:=	FALSE;
	iCompareSeq[ENUM_SeqSM.Once]		:=	60;
END_IF
*)

60:
//Log all the 'gates' - returned from FB_Debounce
FOR uiCounter3	:= 0 TO gc.uiMaxNrDMXTestCh BY 1 DO
	arrxRcvdBufferNPNSeq[uiCounter3]		:= g_ast.arrFBIntNPN[uiCounter3].Q.xGate;
END_FOR
	
iCompareSeq[ENUM_SeqSM.Once]		:=	70;

//IF tonReadWait.Q THEN
//	tonReadWait.IN					:= FALSE;
//Copy hardware state
//	arrxRcvdBufferNPNSeq			:= arrxTestChInputNPN; // linked to hardware
//	arrxRcvdBufferPNPSeq			:= arrxTestChInputPNP; // linked to hardware
//iCompareSeq[ENUM_SeqSM.Once]		:= 90;
//END_IF

70:
//Run Comparos
//Individual
arr_diTestNPNSeqOnceLine[uiLoopRcvIndex]			:= MEMCMP(pBuf1:=ADR(arrxExpctdTmpNPNSeqDMX[uiLoopRcvIndex]),pBuf2:=ADR(arrxRcvdBufferNPNSeq[uiLoopRcvIndex]),n:=SIZEOF(arrxExpctdTmpNPNSeqDMX[uiLoopRcvIndex])); 
//Complete Buffer
arrdiTestNPNSeqOnceComplete[uiLoopRcvIndex]			:= MEMCMP(pBuf1:=ADR(arrxExpctdTmpNPNSeqDMX[cuiMinDUTIndex]),pBuf2:=ADR(arrxRcvdBufferNPNSeq[cuiMinDUTIndex]),n:=gc.uiChannelsUT); 

//log the error index - later

iCompareSeq[ENUM_SeqSM.Once]				:= 80;

80: //Turn off all DMX channels after comparison
FOR uiCounter3 := cuiMinDUTIndex TO gc.uiMaxNrDMXTestCh BY 1 DO
	g_ast.DMX[uiCounter3].IQ.xCmdOff		:= TRUE;
END_FOR

90://Write to DMX hardware, advance state
g_ast.DMXHWOut								:= g_ast.DMXPhysOut;

iCompareSeq[ENUM_SeqSM.Once]				:= 100;

100: //Confirm 'return' to static 
FOR uiCounter3	:= 0 TO gc.uiMaxNrDMXTestCh BY 1 DO
	arrxRcvdBufferNPNSeq[uiCounter3]		:= g_ast.arrFBIntNPN[uiCounter3].Q.xGate;
	IF arrxRcvdBufferNPNSeq[uiCounter3] = arrxExpctdTmpNPNGND[uiCounter3] THEN
		iCompareSeq[ENUM_SeqSM.Once]				:= 110;
	END_IF
END_FOR

110://Write to DMX hardware, advance state
g_ast.DMXHWOut								:= g_ast.DMXPhysOut;

iCompareSeq[ENUM_SeqSM.Once]				:= 120;

